//---------------------------------------------------------------------------------------------------------------
//
//  HAUD 2025.03.31
//
//  - EXAMPLE for top level procedures
//    - transport layer
//    - Collector layer
//    - process layer
//
//  - rewrite/change/discard as you require for your application
//
//  - this function block is NOT intended for direct use outside the scope of this example
//  - maybe the command mechanics are useful for your application
//
//---------------------------------------------------------------------------------------------------------------
FUNCTION_BLOCK fb_Application
VAR
  _eCheck                       : E_APP_CHECK;
  _eInit                        : E_PROGRESS;

  _Ctrl                         : REFERENCE TO ST_APP_CTRL;
  _State                        : REFERENCE TO ST_APP_STATE;

  _eResult                      : E_PROGRESS;

  _eCmd,
  _eCmdOld                      : E_INSTANCE_CMD;
  _eState                       : E_INSTANCE_STATE;

  // Transport Ctrl/State
  _XtsTransportCtrl             : REFERENCE TO ST_XTS_TRANSPORT_CTRL;
  _XtsTransportState            : REFERENCE TO ST_XTS_TRANSPORT_STATE;

  _InstanceCtrl                 : REFERENCE TO ARRAY[1..MAX_PROCESS] OF ST_INSTANCE_CTRL;
  _InstanceState                : REFERENCE TO ARRAY[1..MAX_PROCESS] OF ST_INSTANCE_STATE;
  
  _ItfProcessCollector          : REFERENCE TO ARRAY[1..MAX_PROCESS] OF I_ProcessCollector;

  _ItfProcessList               : REFERENCE TO ARRAY[1..MAX_PROCESS] OF I_Process_LinkedList;

  // timers for this example
  _tonProcess                   : ARRAY[1..MAX_PROCESS] OF Tc2_Standard.TON;
  _tProcess                     : ARRAY[1..MAX_PROCESS] OF TIME;


  _stMsg                        : ST_Message;
  _MessageLevel                 : E_MessageType;

  // ListData()
  _nLoadCaseOld,
  _nLoadCase                    : UINT := 0; // 0 = fully loaded, 2 = mod 5 missing 1, 1 = missing up to 11

  // Work()
  _bSingleOutput                : BOOL;
  _bWriteTimeVariant            : BOOL;
  _nTimeVariant                 : UINT;

  _sAppState                    : STRING;
END_VAR

IF NOT Check() THEN RETURN; END_IF
//-----------------------------------------------------------------------------
//-----------------------------------------------------------------------------
// set message device
//-----------------------------------------------------------------------------
_stMsg.eDevice                  := e_Device.Application;

_eCmd                           := _Ctrl.Cmd;
// check for command change
// get state for cmd
IF (_eCmd <> _eCmdOld)
THEN
  _eState                       := Cmd(_eCmd);
  _eCmdOld                      := _eCmd;
END_IF

CASE _eResult
OF
  E_PROGRESS.PROGRESS_INVALID:
    _State.AppState             := TO_UINT(_eResult);

  E_PROGRESS.PROGRESS_ERROR:
    _State.AppState             := _eState + E_PROGRESS.PROGRESS_ERROR;

  E_PROGRESS.PROGRESS_DONE:
    _State.AppState             := _eState + E_PROGRESS.PROGRESS_DONE;

    IF (_XtsTransportState.GroupInfo.GroupErrorStop) OR
       (_XtsTransportState.GroupInfo.GroupError)     OR
       NOT (_XtsTransportState.XpuInfo.AllPositionsValid)
    THEN
      _eResult                  := E_PROGRESS.PROGRESS_ERROR;
    END_IF
ELSE
  _State.AppState               := _eState + _eResult;

  CASE _eState
  OF
    E_INSTANCE_STATE.INIT:
      _eInit := _eResult        := Init(TRUE);

    E_INSTANCE_STATE.DISABLED:
      _eResult                  := Disable(TRUE);
  
    E_INSTANCE_STATE.ENABLED:
      IF NOT (_XtsTransportState.XpuState.DcLink) OR
         NOT (_XtsTransportState.XpuInfo.AllPositionsValid)
      THEN
        _eResult                := E_PROGRESS.PROGRESS_ERROR;
      ELSE
        _eResult                := Enable(TRUE);
      END_IF

    E_INSTANCE_STATE.WORKING:
      IF NOT (_XtsTransportState.XpuState.DcLink) OR
         NOT (_XtsTransportState.XpuInfo.AllPositionsValid)
      THEN
        _eResult                := E_PROGRESS.PROGRESS_ERROR;
      ELSE
        _eResult                := Work(TRUE);
      END_IF

    E_INSTANCE_STATE.PROCEEDING:
      IF NOT (_XtsTransportState.XpuState.DcLink) OR
         NOT (_XtsTransportState.XpuInfo.AllPositionsValid)
      THEN
        _eResult                := E_PROGRESS.PROGRESS_ERROR;
      ELSE
        _eResult                := Proceed(TRUE);
      END_IF

    E_INSTANCE_STATE.FINISH:
      IF NOT (_XtsTransportState.XpuState.DcLink) OR
         NOT (_XtsTransportState.XpuInfo.AllPositionsValid)
      THEN
        _eResult                := E_PROGRESS.PROGRESS_ERROR;
      ELSE
        _eResult                := Finish(TRUE);
      END_IF

    E_INSTANCE_STATE.CLEARED:
      _eResult                  := Clear(TRUE);


  ELSE
    _eResult                    := E_PROGRESS.PROGRESS_INVALID;
  END_CASE

END_CASE
_State.XtsTransportState        REF= _XtsTransportState;
_State.InstanceStates           REF= _InstanceState;


//IF _bWriteTimeVariant
//THEN
  _bWriteTimeVariant            := FALSE;

  CASE _nTimeVariant
  OF
    0:
      _tProcess[E_INSTANCE.INFEED]           := T#800MS;
      _tProcess[E_INSTANCE.OUTFEED_ROBOT_R1] := T#800MS;
      _tProcess[E_INSTANCE.OUTFEED_ROBOT_R2] := T#800MS;
    1:
      _tProcess[E_INSTANCE.INFEED]           := T#600MS;
      _tProcess[E_INSTANCE.OUTFEED_ROBOT_R1] := T#800MS;
      _tProcess[E_INSTANCE.OUTFEED_ROBOT_R2] := T#800MS;
    2:
      _tProcess[E_INSTANCE.INFEED]           := T#600MS;
      _tProcess[E_INSTANCE.OUTFEED_ROBOT_R1] := T#700MS;
      _tProcess[E_INSTANCE.OUTFEED_ROBOT_R2] := T#700MS;
    3:
      _tProcess[E_INSTANCE.INFEED]           := T#700MS;
      _tProcess[E_INSTANCE.OUTFEED_ROBOT_R1] := T#800MS;
      _tProcess[E_INSTANCE.OUTFEED_ROBOT_R2] := T#800MS;
    4:
      _tProcess[E_INSTANCE.INFEED]           := T#500MS;
      _tProcess[E_INSTANCE.OUTFEED_ROBOT_R1] := T#800MS;
      _tProcess[E_INSTANCE.OUTFEED_ROBOT_R2] := T#800MS;
    5:
      _tProcess[E_INSTANCE.INFEED]           := T#450MS;
      _tProcess[E_INSTANCE.OUTFEED_ROBOT_R1] := T#600MS;
      _tProcess[E_INSTANCE.OUTFEED_ROBOT_R2] := T#600MS;
  ELSE
      _tProcess[E_INSTANCE.INFEED]           := T#800MS;
      _tProcess[E_INSTANCE.OUTFEED_ROBOT_R1] := T#800MS;
      _tProcess[E_INSTANCE.OUTFEED_ROBOT_R2] := T#800MS;
  END_CASE
//END_IF

_sAppState := TO_STRING(_State.AppState);

METHOD Check : BOOL // call this method in the extending/inheriting class
VAR
  _nIdx       : E_INSTANCE;
END_VAR
//-----------------------------------------------------------------------------
//-----------------------------------------------------------------------------
// reference checks
//-----------------------------------------------------------------------------
IF NOT __ISVALIDREF(_Ctrl)
THEN
  _eCheck                   := E_APP_CHECK.INVALID_CTRL_POINTER;
  RETURN;
END_IF

IF NOT __ISVALIDREF(_State)
THEN
  _eCheck                   := E_APP_CHECK.INVALID_STATE_POINTER;
  RETURN;
END_IF

IF NOT __ISVALIDREF(_XtsTransportCtrl)
THEN
  _eCheck                   := E_APP_CHECK.INVALID_TRANSPORT_CTRL_POINTER;
  RETURN;
END_IF

IF NOT __ISVALIDREF(_XtsTransportState)
THEN
  _eCheck                   := E_APP_CHECK.INVALID_TRANSPORT_STATE_POINTER;
  RETURN;
END_IF

IF NOT __ISVALIDREF(_InstanceCtrl)
THEN
  _eCheck                   := E_APP_CHECK.INVALID_INSTANCE_CONTROL_REFERENCE;
  RETURN;
END_IF

IF NOT __ISVALIDREF(_InstanceState)
THEN
  _eCheck                   := E_APP_CHECK.INVALID_INSTANCE_STATE_REFERENCE;
  RETURN;
END_IF
IF NOT __ISVALIDREF(_ItfProcessCollector)
THEN
  _eCheck                   := E_APP_CHECK.INVALID_COLLECTOR_INTERFACE;
  RETURN;
END_IF
IF NOT __ISVALIDREF(_ItfProcessList)
THEN
  _eCheck                   := E_APP_CHECK.INVALID_PROCESS_LIST_INTERFACE;
  RETURN;
END_IF
//-----------------------------------------------------------------------------
//-----------------------------------------------------------------------------
// interface checks
//-----------------------------------------------------------------------------
FOR _nIdx := 1 TO MAX_PROCESS
DO
  IF NOT (_ItfProcessCollector[_nIdx] <> 0) 
  THEN
    _eCheck                 := E_APP_CHECK.INVALID_COLLECTOR_INTERFACE;
    RETURN;
  END_IF
  
  IF NOT (_ItfProcessCollector[_nIdx].ProcessId > 0)
  THEN
    _eCheck                 := E_APP_CHECK.INVALID_PROCESS_LIST_INTERFACE;
    RETURN;
  END_IF
END_FOR
//-----------------------------------------------------------------------------
//-----------------------------------------------------------------------------
_eCheck                     := E_APP_CHECK.CHECK_DONE;
Check                       := TRUE;
END_METHOD

METHOD Clear : E_PROGRESS
VAR_INPUT
  Execute     : BOOL;
END_VAR
VAR_INST
  _nErrorId   : UDINT;
  _eState     : E_PROGRESS;

  _eInstance  : E_INSTANCE;
END_VAR
//-----------------------------------------------------------------------------
IF NOT Execute 
THEN 
	_eState                                         := E_PROGRESS.PROGRESS_INIT; 
END_IF 
//-----------------------------------------------------------------------------
IF NOT Check() 
THEN 
	Clear                                            := E_PROGRESS.PROGRESS_ERROR; 
	RETURN; 
END_IF
//-----------------------------------------------------------------------------
//-----------------------------------------------------------------------------
CASE _eState
OF
  //---------------------------------------------------------------------------------------------------------------
  //---------------------------------------------------------------------------------------------------------------
  E_PROGRESS.PROGRESS_INIT:                   // startup procedure for your application
    IF Execute
    THEN
      ListData(FALSE, TRUE);
      _eState                                             := E_PROGRESS.PROGRESS_BUSY;
  
      FOR _eInstance := E_INSTANCE.BUFFER_INFEED TO E_INSTANCE.SENDER_BUFFER_INFEED
      DO
        _InstanceCtrl[_eInstance].Cmd                     := E_INSTANCE_CMD.NULL;
      END_FOR
  
      IF (_MessageLevel > E_MessageType.eMessageError)
      THEN
        _stMsg.eType                                      := E_MessageType.eMessageInfo;
        _stMsg.eSubdevice                                 := e_Subdevice.Application_Clear;
        _stMsg.iErrorNumber                               := 0;
        _stMsg.sText                                      := concat(TO_STRING(_eState), ': ');
        f_MessageSet(_stMsg);
      END_IF
    END_IF

  //---------------------------------------------------------------------------------------------------------------
  //---------------------------------------------------------------------------------------------------------------
  E_PROGRESS.PROGRESS_BUSY:
    ListData(FALSE, FALSE);
    _InstanceCtrl[E_INSTANCE.BUFFER_INFEED].Cmd           := E_INSTANCE_CMD.INIT;
    //-----------------------------------------------------------------------------------
    CASE _InstanceState[E_INSTANCE.BUFFER_INFEED].State
    OF
      E_INSTANCE_STATE.DISABLED:
        CASE _InstanceState[E_INSTANCE.BUFFER_INFEED].Progress
        OF
          E_PROGRESS.PROGRESS_BUSY:           // check for startup to be done
            _InstanceCtrl[E_INSTANCE.BUFFER_INFEED].Cmd   := E_INSTANCE_CMD.DISABLE;
            _eState                                       := E_PROGRESS.PROGRESS_PREPARE; // go check next insatnce

            IF (_MessageLevel > E_MessageType.eMessageError)
            THEN
              _stMsg.eType          := E_MessageType.eMessageInfo;
              _stMsg.eSubdevice     := e_Subdevice.Application_Clear;
              _stMsg.iErrorNumber   := 0;
              _stMsg.sText          := concat(TO_STRING(E_INSTANCE.BUFFER_INFEED), ': cleared');
              f_MessageSet(_stMsg);
            END_IF
        END_CASE
    END_CASE

  //---------------------------------------------------------------------------------------------------------------
  //---------------------------------------------------------------------------------------------------------------
  E_PROGRESS.PROGRESS_PREPARE:
    _InstanceCtrl[E_INSTANCE.INFEED].Cmd                  := E_INSTANCE_CMD.INIT;
    //-----------------------------------------------------------------------------------
    CASE _InstanceState[E_INSTANCE.INFEED].State
    OF
      E_INSTANCE_STATE.DISABLED:
        CASE _InstanceState[E_INSTANCE.INFEED].Progress
        OF
          E_PROGRESS.PROGRESS_BUSY:           // check for startup to be done
          _InstanceCtrl[E_INSTANCE.INFEED].Cmd            := E_INSTANCE_CMD.DISABLE;
          _eState                                         := E_PROGRESS.PROGRESS_STARTUP; // go check next insatnce

          IF (_MessageLevel > E_MessageType.eMessageError)
          THEN
            _stMsg.eType          := E_MessageType.eMessageInfo;
            _stMsg.eSubdevice     := e_Subdevice.Application_Clear;
            _stMsg.iErrorNumber   := 0;
            _stMsg.sText          := concat(TO_STRING(E_INSTANCE.INFEED), ': cleared');
            f_MessageSet(_stMsg);
          END_IF
        END_CASE
    END_CASE

  //---------------------------------------------------------------------------------------------------------------
  //---------------------------------------------------------------------------------------------------------------
  E_PROGRESS.PROGRESS_STARTUP:
    _InstanceCtrl[E_INSTANCE.BUFFER_OUTFEED].Cmd    := E_INSTANCE_CMD.INIT;
    //-----------------------------------------------------------------------------------
    CASE _InstanceState[E_INSTANCE.BUFFER_OUTFEED].State
    OF
      E_INSTANCE_STATE.DISABLED:
        CASE _InstanceState[E_INSTANCE.BUFFER_OUTFEED].Progress
        OF
          E_PROGRESS.PROGRESS_BUSY:           // check for startup to be done
          _InstanceCtrl[E_INSTANCE.BUFFER_OUTFEED].Cmd   := E_INSTANCE_CMD.DISABLE;
          _eState                                         := E_PROGRESS.PROGRESS_CHECK; // go check next insatnce

          IF (_MessageLevel > E_MessageType.eMessageError)
          THEN
            _stMsg.eType          := E_MessageType.eMessageInfo;
            _stMsg.eSubdevice     := e_Subdevice.Application_Clear;
            _stMsg.iErrorNumber   := 0;
            _stMsg.sText          := concat(TO_STRING(E_INSTANCE.BUFFER_OUTFEED), ': cleared');
            f_MessageSet(_stMsg);
          END_IF
        END_CASE
    END_CASE

  //---------------------------------------------------------------------------------------------------------------
  //---------------------------------------------------------------------------------------------------------------
  E_PROGRESS.PROGRESS_CHECK:
    _InstanceCtrl[E_INSTANCE.OUTFEED_ROBOT_R1].Cmd        := E_INSTANCE_CMD.INIT;
    //-----------------------------------------------------------------------------------
    CASE _InstanceState[E_INSTANCE.OUTFEED_ROBOT_R1].State
    OF
      E_INSTANCE_STATE.DISABLED:
        CASE _InstanceState[E_INSTANCE.OUTFEED_ROBOT_R1].Progress
        OF
          E_PROGRESS.PROGRESS_BUSY:           // check for startup to be done
          _InstanceCtrl[E_INSTANCE.OUTFEED_ROBOT_R1].Cmd  := E_INSTANCE_CMD.DISABLE;
          _eState                                         := E_PROGRESS.PROGRESS_OCCUPIED; // go check next insatnce

          IF (_MessageLevel > E_MessageType.eMessageError)
          THEN
            _stMsg.eType          := E_MessageType.eMessageInfo;
            _stMsg.eSubdevice     := e_Subdevice.Application_Clear;
            _stMsg.iErrorNumber   := 0;
            _stMsg.sText          := concat(TO_STRING(E_INSTANCE.OUTFEED_ROBOT_R1), ': cleared');
            f_MessageSet(_stMsg);
          END_IF
        END_CASE
    END_CASE

  //---------------------------------------------------------------------------------------------------------------
  //---------------------------------------------------------------------------------------------------------------
  E_PROGRESS.PROGRESS_OCCUPIED:
    _InstanceCtrl[E_INSTANCE.OUTFEED_ROBOT_R2].Cmd        := E_INSTANCE_CMD.INIT;
    //-----------------------------------------------------------------------------------
    CASE _InstanceState[E_INSTANCE.OUTFEED_ROBOT_R2].State
    OF
      E_INSTANCE_STATE.DISABLED:
        CASE _InstanceState[E_INSTANCE.OUTFEED_ROBOT_R2].Progress
        OF
          E_PROGRESS.PROGRESS_BUSY:           // check for startup to be done
          _InstanceCtrl[E_INSTANCE.OUTFEED_ROBOT_R2].Cmd  := E_INSTANCE_CMD.DISABLE;
          _eState                                         := E_PROGRESS.PROGRESS_WORKING; // go check next insatnce

          IF (_MessageLevel > E_MessageType.eMessageError)
          THEN
            _stMsg.eType          := E_MessageType.eMessageInfo;
            _stMsg.eSubdevice     := e_Subdevice.Application_Clear;
            _stMsg.iErrorNumber   := 0;
            _stMsg.sText          := concat(TO_STRING(E_INSTANCE.OUTFEED_ROBOT_R2), ': cleared');
            f_MessageSet(_stMsg);
          END_IF
        END_CASE
    END_CASE

  //---------------------------------------------------------------------------------------------------------------
  //---------------------------------------------------------------------------------------------------------------
  E_PROGRESS.PROGRESS_WORKING:
    _InstanceCtrl[E_INSTANCE.SENDER_FAST].Cmd             := E_INSTANCE_CMD.INIT;
    //-----------------------------------------------------------------------------------
    CASE _InstanceState[E_INSTANCE.SENDER_FAST].State
    OF
      E_INSTANCE_STATE.DISABLED:
        CASE _InstanceState[E_INSTANCE.SENDER_FAST].Progress
        OF
          E_PROGRESS.PROGRESS_BUSY:           // check for startup to be done
          _InstanceCtrl[E_INSTANCE.SENDER_FAST].Cmd       := E_INSTANCE_CMD.DISABLE;
          _eState                                         := E_PROGRESS.PROGRESS_STILL_WORKING; // go check next insatnce

          IF (_MessageLevel > E_MessageType.eMessageError)
          THEN
            _stMsg.eType          := E_MessageType.eMessageInfo;
            _stMsg.eSubdevice     := e_Subdevice.Application_Clear;
            _stMsg.iErrorNumber   := 0;
            _stMsg.sText          := concat(TO_STRING(E_INSTANCE.SENDER_FAST), ': cleared');
            f_MessageSet(_stMsg);
          END_IF
        END_CASE
    END_CASE

  //---------------------------------------------------------------------------------------------------------------
  //---------------------------------------------------------------------------------------------------------------
  E_PROGRESS.PROGRESS_STILL_WORKING:
    _InstanceCtrl[E_INSTANCE.SENDER_BUFFER_INFEED].Cmd    := E_INSTANCE_CMD.INIT;
    //-----------------------------------------------------------------------------------
    CASE _InstanceState[E_INSTANCE.SENDER_BUFFER_INFEED].State
    OF
      E_INSTANCE_STATE.DISABLED:
        CASE _InstanceState[E_INSTANCE.SENDER_BUFFER_INFEED].Progress
        OF
          E_PROGRESS.PROGRESS_BUSY:           // check for startup to be done
          _InstanceCtrl[E_INSTANCE.SENDER_BUFFER_INFEED].Cmd    := E_INSTANCE_CMD.DISABLE;
          _eState                                         := E_PROGRESS.PROGRESS_DONE;

          IF (_MessageLevel > E_MessageType.eMessageError)
          THEN
            _stMsg.eType          := E_MessageType.eMessageInfo;
            _stMsg.eSubdevice     := e_Subdevice.Application_Clear;
            _stMsg.iErrorNumber   := 0;
            _stMsg.sText          := concat(TO_STRING(E_INSTANCE.SENDER_BUFFER_INFEED), ': cleared');
            f_MessageSet(_stMsg);
          END_IF

          IF (_MessageLevel > E_MessageType.eMessageError)
          THEN
            _stMsg.eType          := E_MessageType.eMessageInfo;
            _stMsg.eSubdevice     := e_Subdevice.Application_Clear;
            _stMsg.iErrorNumber   := 0;
            _stMsg.sText          := concat(TO_STRING(_eState), ': ');
            f_MessageSet(_stMsg);
          END_IF
        END_CASE
    END_CASE
END_CASE
//-----------------------------------------------------------------------------
//-----------------------------------------------------------------------------

Clear                                              := _eState;
END_METHOD

METHOD PRIVATE Cmd : E_INSTANCE_STATE
VAR_INPUT
  Command   : E_INSTANCE_CMD;
END_VAR
VAR_INST
  _eRslt    : E_PROGRESS;
  _eState   : E_INSTANCE_STATE;
END_VAR
IF NOT Check() THEN RETURN; END_IF


CASE Command
OF
  E_INSTANCE_CMD.NULL:  // clear all method calls
    _eState               := E_INSTANCE_STATE.NULL;
    _eRslt                := Init    (FALSE);
    _eRslt                := Disable (FALSE);
    _eRslt                := Enable  (FALSE);
    _eRslt                := Work    (FALSE);
    _eRslt                := Proceed (FALSE);
    _eRslt                := Finish  (FALSE);
    _eRslt                := Clear   (FALSE);

  E_INSTANCE_CMD.INIT:  // clear methods for initialization
    _eState               := E_INSTANCE_STATE.INIT;
    _eResult              := Init(FALSE);

ELSE
  IF NOT (_eInit = E_PROGRESS.PROGRESS_DONE)
  THEN
    // no init, no further commands possible
    _eState               := E_INSTANCE_STATE.INVALID;
  ELSE
    CASE Command
    OF
      E_INSTANCE_CMD.DISABLE:
        _eState           := E_INSTANCE_STATE.DISABLED;
        _eResult          := Disable (FALSE);

      E_INSTANCE_CMD.ENABLE:
        _eState           := E_INSTANCE_STATE.ENABLED;
        _eResult          := Enable  (FALSE);

      E_INSTANCE_CMD.WORK:
        _eState           := E_INSTANCE_STATE.WORKING;
        _eResult          := Work    (FALSE);

      E_INSTANCE_CMD.PROCEED:
        _eState           := E_INSTANCE_STATE.PROCEEDING;
        _eResult          := Proceed (FALSE);

      E_INSTANCE_CMD.FINISH:
        _eState           := E_INSTANCE_STATE.FINISH;
        _eResult          := Finish  (FALSE);

      E_INSTANCE_CMD.CLEAR:
        _eState           := E_INSTANCE_STATE.CLEARED;
        _eResult          := Clear   (FALSE);

    ELSE
        _eState           := E_INSTANCE_STATE.INVALID;
    END_CASE
  END_IF
END_CASE

Cmd                       := _eState;
END_METHOD

PROPERTY CollectorInterface : REFERENCE TO ARRAY[1..MAX_PROCESS] OF I_ProcessCollector
SET
_ItfProcessCollector REF= CollectorInterface;
END_SET
END_PROPERTY

PROPERTY Ctrl : REFERENCE TO ST_APP_CTRL
SET
_Ctrl REF= Ctrl;
END_SET
END_PROPERTY

METHOD Disable : E_PROGRESS // RemoveAllAxis from CA Group, disable CA Group, disable all movers
VAR_INPUT
  Execute     : BOOL;
END_VAR
VAR_INST
  _nErrorId   : UDINT;
  _eState     : E_PROGRESS;
END_VAR
//-----------------------------------------------------------------------------
IF NOT Execute 
THEN 
	_eState                       := E_PROGRESS.PROGRESS_INIT; 
END_IF 
//-----------------------------------------------------------------------------
IF NOT Check() 
THEN 
	Disable                       := E_PROGRESS.PROGRESS_ERROR; 
	RETURN; 
END_IF
//-----------------------------------------------------------------------------
//-----------------------------------------------------------------------------
CASE _eState
OF
  E_PROGRESS.PROGRESS_INIT:
    IF Execute
    THEN
      _nErrorId                 := 0;

      _XtsTransportCtrl.Cmd     := E_XTS_TRANSPORT_CTRL.CMD_NULL;
      _eState                   := E_PROGRESS.PROGRESS_BUSY;

      IF (_MessageLevel > E_MessageType.eMessageError)
      THEN
        _stMsg.eType            := E_MessageType.eMessageInfo;
        _stMsg.eSubdevice       := e_Subdevice.Application_Disable;
        _stMsg.iErrorNumber     := 0;
        _stMsg.sText            := concat(TO_STRING(_eState), ': ');
        f_MessageSet(_stMsg);
      END_IF
    END_IF

  E_PROGRESS.PROGRESS_BUSY:
    _XtsTransportCtrl.Cmd       := E_XTS_TRANSPORT_CTRL.CMD_GROUP_CLEAR; 
    _eState                     := E_PROGRESS.PROGRESS_PREPARE;
END_CASE
//-----------------------------------------------------------------------------
//-----------------------------------------------------------------------------
CASE _eState
OF
  E_PROGRESS.PROGRESS_PREPARE:
    IF (_XtsTransportState.State = E_XTS_TRANSPORT_STATE.TRANSPORT_GROUP_CLEAR + E_PROGRESS.PROGRESS_ERROR)
    THEN
      _eState                   := E_PROGRESS.PROGRESS_BUSY;
      _XtsTransportCtrl.Cmd     := E_XTS_TRANSPORT_CTRL.CMD_NULL;

      _nErrorId                 := _XtsTransportState.GroupInfo.GroupErrorId; 

    ELSIF (_XtsTransportState.State = E_XTS_TRANSPORT_STATE.TRANSPORT_GROUP_CLEAR + E_PROGRESS.PROGRESS_DONE)
    THEN
      _eState                   := E_PROGRESS.PROGRESS_STARTUP;

    END_IF
END_CASE
//-----------------------------------------------------------------------------
//-----------------------------------------------------------------------------
CASE _eState
OF
  E_PROGRESS.PROGRESS_STARTUP:
    _XtsTransportCtrl.Cmd       := E_XTS_TRANSPORT_CTRL.CMD_MOVER_DISABLE; 
    _eState                     := E_PROGRESS.PROGRESS_CHECK;
END_CASE
//-----------------------------------------------------------------------------
//-----------------------------------------------------------------------------
CASE _eState
OF
  E_PROGRESS.PROGRESS_CHECK:
    IF (_XtsTransportState.State = E_XTS_TRANSPORT_STATE.TRANSPORT_MOVER_DISABLE + E_PROGRESS.PROGRESS_ERROR)
    THEN
      _eState                   := E_PROGRESS.PROGRESS_ERROR;

    ELSIF (_XtsTransportState.State = E_XTS_TRANSPORT_STATE.TRANSPORT_MOVER_DISABLE + E_PROGRESS.PROGRESS_DONE)
    THEN
      _eState                   := E_PROGRESS.PROGRESS_DONE;

      IF (_MessageLevel > E_MessageType.eMessageError)
      THEN
        _stMsg.eType            := E_MessageType.eMessageInfo;
        _stMsg.eSubdevice       := e_Subdevice.Application_Disable;
        _stMsg.iErrorNumber     := 0;
        _stMsg.sText            := concat(TO_STRING(_eState), ': ');
        f_MessageSet(_stMsg);
      END_IF
    END_IF
END_CASE
//-----------------------------------------------------------------------------
//-----------------------------------------------------------------------------

Disable                         := _eState;
END_METHOD

METHOD Enable : E_PROGRESS // AddAllAxis to CA Group, Enable CA Group, Enable all movers
VAR_INPUT
  Execute     : BOOL;
END_VAR
VAR_INST
  _nErrorId   : UDINT;
  _eState     : E_PROGRESS;
END_VAR
//-----------------------------------------------------------------------------
IF NOT Execute 
THEN 
	_eState                       := E_PROGRESS.PROGRESS_INIT; 
END_IF 
//-----------------------------------------------------------------------------
IF NOT Check() 
THEN 
	Enable                        := E_PROGRESS.PROGRESS_ERROR; 
	RETURN; 
END_IF
//-----------------------------------------------------------------------------
//-----------------------------------------------------------------------------
CASE _eState
OF
  E_PROGRESS.PROGRESS_INIT:
    IF Execute
    THEN

      IF (GVL_APPLICATION.bOutput_R1R2)
      THEN
        MAIN_APP.ProcessInit_R1R2();
      ELSE
        MAIN_APP.ProcessInit_CLAMP();
      END_IF

      _nErrorId                 := 0;

      _XtsTransportCtrl.Cmd     := E_XTS_TRANSPORT_CTRL.CMD_NULL;
      _eState                   := E_PROGRESS.PROGRESS_BUSY;

      IF (_MessageLevel > E_MessageType.eMessageError)
      THEN
        _stMsg.eType            := E_MessageType.eMessageInfo;
        _stMsg.eSubdevice       := e_Subdevice.Application_Enable;
        _stMsg.iErrorNumber     := 0;
        _stMsg.sText            := concat(TO_STRING(_eState), ': ');
        f_MessageSet(_stMsg);
      END_IF
    END_IF

  E_PROGRESS.PROGRESS_BUSY:
    _XtsTransportCtrl.Cmd       := E_XTS_TRANSPORT_CTRL.CMD_GROUP_BUILD; 
    _eState                     := E_PROGRESS.PROGRESS_PREPARE;
END_CASE
//-----------------------------------------------------------------------------
//-----------------------------------------------------------------------------
CASE _eState
OF
  E_PROGRESS.PROGRESS_PREPARE:
    IF (_XtsTransportState.State = E_XTS_TRANSPORT_STATE.TRANSPORT_GROUP_BUILD + E_PROGRESS.PROGRESS_ERROR)
    THEN
      _eState                   := E_PROGRESS.PROGRESS_ERROR;
      _nErrorId                 := _XtsTransportState.GroupInfo.GroupErrorId; 

    ELSIF (_XtsTransportState.State = E_XTS_TRANSPORT_STATE.TRANSPORT_GROUP_BUILD + E_PROGRESS.PROGRESS_DONE)
    THEN
      _eState                   := E_PROGRESS.PROGRESS_STARTUP;
    END_IF
END_CASE
//-----------------------------------------------------------------------------
//-----------------------------------------------------------------------------
CASE _eState
OF
  E_PROGRESS.PROGRESS_STARTUP:
    _XtsTransportCtrl.Cmd       := E_XTS_TRANSPORT_CTRL.CMD_MOVER_ENABLE; 
    _eState                     := E_PROGRESS.PROGRESS_CHECK;
END_CASE
//-----------------------------------------------------------------------------
//-----------------------------------------------------------------------------
CASE _eState
OF
  E_PROGRESS.PROGRESS_CHECK:
    IF (_XtsTransportState.State = E_XTS_TRANSPORT_STATE.TRANSPORT_MOVER_ENABLE + E_PROGRESS.PROGRESS_ERROR)
    THEN
      _eState                   := E_PROGRESS.PROGRESS_ERROR;

    ELSIF (_XtsTransportState.State = E_XTS_TRANSPORT_STATE.TRANSPORT_MOVER_ENABLE + E_PROGRESS.PROGRESS_DONE)
    THEN
      _eState                   := E_PROGRESS.PROGRESS_OCCUPIED;
    END_IF
END_CASE
//-----------------------------------------------------------------------------
//-----------------------------------------------------------------------------
CASE _eState
OF
  E_PROGRESS.PROGRESS_OCCUPIED:
    _XtsTransportCtrl.Cmd       := E_XTS_TRANSPORT_CTRL.CMD_GROUP_ENABLE; 
    _eState                     := E_PROGRESS.PROGRESS_WORKING;
END_CASE
//-----------------------------------------------------------------------------
//-----------------------------------------------------------------------------
CASE _eState
OF
  E_PROGRESS.PROGRESS_WORKING:
    IF (_XtsTransportState.State = E_XTS_TRANSPORT_STATE.TRANSPORT_GROUP_ENABLE + E_PROGRESS.PROGRESS_ERROR)
    THEN
      _eState                   := E_PROGRESS.PROGRESS_ERROR;

    ELSIF (_XtsTransportState.State = E_XTS_TRANSPORT_STATE.TRANSPORT_GROUP_ENABLE + E_PROGRESS.PROGRESS_DONE)
    THEN
      _eState                   := E_PROGRESS.PROGRESS_DONE;

      IF (_MessageLevel > E_MessageType.eMessageError)
      THEN
        _stMsg.eType            := E_MessageType.eMessageInfo;
        _stMsg.eSubdevice       := e_Subdevice.Application_Enable;
        _stMsg.iErrorNumber     := 0;
        _stMsg.sText            := concat(TO_STRING(_eState), ': ');
        f_MessageSet(_stMsg);
      END_IF
    END_IF
END_CASE
//-----------------------------------------------------------------------------
//-----------------------------------------------------------------------------

Enable                          := _eState;
END_METHOD

METHOD Finish : E_PROGRESS
VAR_INPUT
  Execute     : BOOL;
END_VAR
VAR_INST
  _nErrorId               : UDINT;
  _eState                 : E_PROGRESS;

  _nExp                   : BYTE;
  _WriteData              : ST_PROCESS_DATA;
  _ListResult             : ST_PROCESS_LIST_RESULT;

  _eInst                  : E_INSTANCE;
  _bDbg : BOOL;
  {attribute 'displaymode':='bin'}
  _wDisable               : T_PROCESS;

  _nSwitch                : UINT;
  _TransportState         : E_XTS_TRANSPORT_STATE;
  _JobResult              : E_PROGRESS;
END_VAR
//-----------------------------------------------------------------------------
IF NOT Execute 
THEN 
	_eState                       := E_PROGRESS.PROGRESS_INIT; 
END_IF 
//-----------------------------------------------------------------------------
IF NOT Check() 
THEN 
	Finish                        := E_PROGRESS.PROGRESS_ERROR; 
	RETURN; 
END_IF
//-----------------------------------------------------------------------------
//-----------------------------------------------------------------------------
CASE _eState
OF
  E_PROGRESS.PROGRESS_INIT:
    IF Execute
    THEN
      _nErrorId                 := 0;
      _JobResult                := ListData(TRUE, FALSE);     // reset simulated transfersystem

      IF NOT (_XtsTransportState.GroupInfo.GroupErrorStop)
      THEN
        _eState                 := E_PROGRESS.PROGRESS_BUSY;

        IF (_MessageLevel > E_MessageType.eMessageError)
        THEN
          _stMsg.eType          := E_MessageType.eMessageInfo;
          _stMsg.eSubdevice     := e_Subdevice.Application_Finish;
          _stMsg.iErrorNumber   := 0;
          _stMsg.sText          := concat(TO_STRING(_eState), ': ');
          f_MessageSet(_stMsg);
        END_IF
      ELSE
        _nErrorId               := _XtsTransportState.GroupInfo.GroupErrorId;
        _eState                 := E_PROGRESS.PROGRESS_ERROR;

        _stMsg.eType            := E_MessageType.eMessageError;
        _stMsg.eSubdevice       := e_Subdevice.Application_Finish;
        _stMsg.iErrorNumber     := _nErrorId;
        _stMsg.sText            := concat(TO_STRING(_eState), ': ');
        _stMsg.sText            := concat(_stMsg.sText, ' CaGroup ErrorStop');
        f_MessageSet(_stMsg);
      END_IF
    END_IF


  E_PROGRESS.PROGRESS_BUSY:
    IF (_XtsTransportState.State = E_XTS_TRANSPORT_STATE.TRANSPORT_START   + E_PROGRESS.PROGRESS_ERROR) OR
       (_XtsTransportState.State = E_XTS_TRANSPORT_STATE.TRANSPORT_RESTART + E_PROGRESS.PROGRESS_ERROR)
    THEN
      _eState                   := E_PROGRESS.PROGRESS_ERROR;

      _stMsg.eType              := E_MessageType.eMessageError;
      _stMsg.eSubdevice         := e_Subdevice.Application_Finish;
      _stMsg.iErrorNumber       := 0;
      _stMsg.sText              := concat(TO_STRING(_eState), ': ');
      _stMsg.sText              := concat(_stMsg.sText, TO_STRING(_XtsTransportState.State MOD E_PROGRESS.PROGRESS_ERROR));
      f_MessageSet(_stMsg);

    ELSIF (_XtsTransportState.State = E_XTS_TRANSPORT_STATE.TRANSPORT_START   + E_PROGRESS.PROGRESS_DONE) OR
          (_XtsTransportState.State = E_XTS_TRANSPORT_STATE.TRANSPORT_RESTART + E_PROGRESS.PROGRESS_DONE)
    THEN
      _JobResult                := ListData(FALSE, FALSE);     // stop simulated transfersystem
      _wDisable                 := 0;
      _eState                   := E_PROGRESS.PROGRESS_PREPARE;

      IF (_MessageLevel > E_MessageType.eMessageError)
      THEN
        _stMsg.eType            := E_MessageType.eMessageInfo;
        _stMsg.eSubdevice       := e_Subdevice.Application_Finish;
        _stMsg.iErrorNumber     := 0;
        _stMsg.sText            := concat(TO_STRING(_eState), ': ');
        _stMsg.sText            := concat(_stMsg.sText, TO_STRING(_XtsTransportState.State MOD E_PROGRESS.PROGRESS_DONE));
        f_MessageSet(_stMsg);
      END_IF
    END_IF
END_CASE
//-----------------------------------------------------------------------------
//-----------------------------------------------------------------------------
CASE _eState
OF
  E_PROGRESS.PROGRESS_PREPARE:  // SENDER_BUFFER_INFEED sends movers to BUFFER_INFEED
                                //  - this instance has to stop first
    CASE _InstanceState[E_INSTANCE.SENDER_BUFFER_INFEED].State
    OF
    E_INSTANCE_STATE.DISABLED:

      CASE _InstanceState[E_INSTANCE.SENDER_BUFFER_INFEED].Progress
      OF
      E_PROGRESS.PROGRESS_BUSY,
      E_PROGRESS.PROGRESS_PREPARE:
        _eState                                               := E_PROGRESS.PROGRESS_STARTUP;
        _InstanceCtrl[E_INSTANCE.SENDER_BUFFER_INFEED].Cmd    := E_INSTANCE_CMD.DISABLE;
  
        _wDisable                                             := _ItfProcessCollector[E_INSTANCE.SENDER_BUFFER_INFEED].
                                                                 SetBit(_wDisable, TO_BYTE(E_INSTANCE.SENDER_BUFFER_INFEED-1));
        IF (_MessageLevel > E_MessageType.eMessageError)
        THEN
          _stMsg.eType                                        := E_MessageType.eMessageInfo;
          _stMsg.eSubdevice                                   := e_Subdevice.Application_Finish;
          _stMsg.iErrorNumber                                 := 0;
          _stMsg.sText                                        := concat(TO_STRING(E_INSTANCE.SENDER_BUFFER_INFEED), ': _wDisable  ');
          _stMsg.sText                                        := concat(_stMsg.sText, _ItfProcessCollector[E_INSTANCE.SENDER_BUFFER_INFEED].BitsToString(_wDisable));
          f_MessageSet(_stMsg);
        END_IF
      END_CASE
    END_CASE
END_CASE
//-----------------------------------------------------------------------------
//-----------------------------------------------------------------------------
CASE _eState
OF
  E_PROGRESS.PROGRESS_STARTUP:
    _JobResult                                                := ListData(FALSE, FALSE);     // stop simulated transfersystem

    CASE _InstanceState[E_INSTANCE.BUFFER_INFEED].State
    OF
    E_INSTANCE_STATE.DISABLED,
    E_INSTANCE_STATE.DETECTION:

      _eState                                                 := E_PROGRESS.PROGRESS_CHECK;
      _InstanceCtrl[E_INSTANCE.BUFFER_INFEED].Cmd             := E_INSTANCE_CMD.DISABLE;
  
      IF NOT (_ItfProcessCollector[E_INSTANCE.BUFFER_INFEED].GetBit(_wDisable, TO_BYTE(E_INSTANCE.BUFFER_INFEED-1)))
      THEN
        _wDisable                                             := _ItfProcessCollector[E_INSTANCE.BUFFER_INFEED].
                                                                 SetBit(_wDisable, TO_BYTE(E_INSTANCE.BUFFER_INFEED-1));
  
        IF (_MessageLevel > E_MessageType.eMessageError)
        THEN
          _stMsg.eType                                        := E_MessageType.eMessageInfo;
          _stMsg.eSubdevice                                   := e_Subdevice.Application_Finish;
          _stMsg.iErrorNumber                                 := 0;
          _stMsg.sText                                        := concat(TO_STRING(E_INSTANCE.BUFFER_INFEED), ': _wDisable  ');
          _stMsg.sText                                        := concat(_stMsg.sText, _ItfProcessCollector[E_INSTANCE.BUFFER_INFEED].BitsToString(_wDisable));
          f_MessageSet(_stMsg);
        END_IF
      END_IF

    E_INSTANCE_STATE.ENABLED:
      _InstanceCtrl[E_INSTANCE.BUFFER_INFEED].Cmd             := E_INSTANCE_CMD.DISABLE;


    E_INSTANCE_STATE.FINISH:
      CASE _InstanceState[E_INSTANCE.BUFFER_INFEED].Progress
      OF
        E_PROGRESS.PROGRESS_BUSY:
          _InstanceCtrl[E_INSTANCE.BUFFER_INFEED].Cmd         := E_INSTANCE_CMD.FINISH;

        E_PROGRESS.PROGRESS_OCCUPIED:
          _InstanceCtrl[E_INSTANCE.BUFFER_INFEED].Cmd         := E_INSTANCE_CMD.PROCEED;
      END_CASE
    END_CASE
END_CASE
//-----------------------------------------------------------------------------
//-----------------------------------------------------------------------------
CASE _eState
OF
  E_PROGRESS.PROGRESS_CHECK:
    CASE _InstanceState[E_INSTANCE.INFEED].State
    OF
    E_INSTANCE_STATE.DISABLED,
    E_INSTANCE_STATE.DETECTION:

      CASE _InstanceState[E_INSTANCE.INFEED].Progress
      OF
      E_PROGRESS.PROGRESS_BUSY:
          IF (_ItfProcessCollector[E_INSTANCE.BUFFER_INFEED].QueueProcessCount > 0)
          THEN
            _eState                                           := E_PROGRESS.PROGRESS_STARTUP;
            _InstanceCtrl[E_INSTANCE.INFEED].Cmd              := E_INSTANCE_CMD.ENABLE;

          ELSIF (_ItfProcessList[E_INSTANCE.INFEED].Count > 0)
          THEN
            _InstanceCtrl[E_INSTANCE.INFEED].Cmd              := E_INSTANCE_CMD.ENABLE;
          ELSE
            _eState                                           := E_PROGRESS.PROGRESS_OCCUPIED;
            _InstanceCtrl[E_INSTANCE.INFEED].Cmd              := E_INSTANCE_CMD.DISABLE;

            IF NOT (_ItfProcessCollector[E_INSTANCE.INFEED].GetBit(_wDisable, TO_BYTE(E_INSTANCE.INFEED-1)))
            THEN
              _wDisable                                       := _ItfProcessCollector[E_INSTANCE.INFEED].
                                                                   SetBit(_wDisable, TO_BYTE(E_INSTANCE.INFEED-1));

              IF (_MessageLevel > E_MessageType.eMessageError)
              THEN
                _stMsg.eType                                  := E_MessageType.eMessageInfo;
                _stMsg.eSubdevice                             := e_Subdevice.Application_Finish;
                _stMsg.iErrorNumber                           := 0;
                _stMsg.sText                                  := concat(TO_STRING(E_INSTANCE.INFEED), ': _wDisable ');
                _stMsg.sText                                  := concat(_stMsg.sText, _ItfProcessCollector[E_INSTANCE.INFEED].BitsToString(_wDisable));
                f_MessageSet(_stMsg);
              END_IF
            END_IF
          END_IF
      END_CASE

    E_INSTANCE_STATE.ENABLED:
      CASE _InstanceState[E_INSTANCE.INFEED].Progress
      OF
        E_PROGRESS.PROGRESS_OCCUPIED:
          _InstanceCtrl[E_INSTANCE.INFEED].Cmd                := E_INSTANCE_CMD.PROCEED;
      END_CASE


    E_INSTANCE_STATE.WORKING:
      CASE _InstanceState[E_INSTANCE.INFEED].Progress
      OF
        E_PROGRESS.PROGRESS_BUSY:
          _InstanceCtrl[E_INSTANCE.INFEED].Cmd                := E_INSTANCE_CMD.WORK;
          _tonProcess [E_INSTANCE.INFEED]
                                          (IN                 := FALSE, 
                                           PT                 := _tProcess[E_INSTANCE.INFEED]);
  
        E_PROGRESS.PROGRESS_CHECK:
          _tonProcess [E_INSTANCE.INFEED]
                                          (IN                 := TRUE, 
                                           PT                 := _tProcess[E_INSTANCE.INFEED]);
  
          IF _tonProcess [E_INSTANCE.INFEED].Q
          THEN
            _InstanceCtrl[E_INSTANCE.INFEED].Cmd              := E_INSTANCE_CMD.FINISH;
          END_IF
      END_CASE

    E_INSTANCE_STATE.FINISH:
      CASE _InstanceState[E_INSTANCE.INFEED].Progress
      OF
        E_PROGRESS.PROGRESS_BUSY:
          _InstanceCtrl[E_INSTANCE.INFEED].Cmd                := E_INSTANCE_CMD.FINISH;

        E_PROGRESS.PROGRESS_OCCUPIED:
          _InstanceCtrl[E_INSTANCE.INFEED].Cmd                := E_INSTANCE_CMD.PROCEED;
      END_CASE
    END_CASE

    CASE _InstanceState[E_INSTANCE.BUFFER_OUTFEED].State
    OF
    E_INSTANCE_STATE.DISABLED:

      CASE _InstanceState[E_INSTANCE.BUFFER_OUTFEED].Progress
      OF
      E_PROGRESS.PROGRESS_BUSY:
        _InstanceCtrl[E_INSTANCE.BUFFER_OUTFEED].Cmd    := E_INSTANCE_CMD.ENABLE;
      END_CASE

    E_INSTANCE_STATE.FINISH:
      CASE _InstanceState[E_INSTANCE.BUFFER_OUTFEED].Progress
      OF
        E_PROGRESS.PROGRESS_BUSY:
          _InstanceCtrl[E_INSTANCE.BUFFER_OUTFEED].Cmd  := E_INSTANCE_CMD.FINISH;

        E_PROGRESS.PROGRESS_OCCUPIED:
          _InstanceCtrl[E_INSTANCE.BUFFER_OUTFEED].Cmd  := E_INSTANCE_CMD.PROCEED;

        E_PROGRESS.PROGRESS_DONE:
          _InstanceCtrl[E_INSTANCE.BUFFER_OUTFEED].Cmd  := E_INSTANCE_CMD.DISABLE;
      END_CASE
    END_CASE

    CASE _InstanceState[E_INSTANCE.SENDER_FAST].State
    OF
      E_INSTANCE_STATE.DISABLED:
        CASE _InstanceState[E_INSTANCE.SENDER_FAST].Progress
        OF
          E_PROGRESS.PROGRESS_BUSY:
            IF NOT (_ItfProcessCollector[E_INSTANCE.OUTFEED_ROBOT_R1].QueueProcessCount < 12) OR 
               NOT (_ItfProcessCollector[E_INSTANCE.OUTFEED_ROBOT_R2].QueueProcessCount < 12)
            THEN
              _InstanceCtrl[E_INSTANCE.SENDER_FAST].Cmd       := E_INSTANCE_CMD.ENABLE;

            ELSIF (_ItfProcessCollector[E_INSTANCE.SENDER_FAST].QueueProcessCount > 0)
            THEN
              _InstanceCtrl[E_INSTANCE.SENDER_FAST].Cmd       := E_INSTANCE_CMD.ENABLE;
            ELSE
              _InstanceCtrl[E_INSTANCE.SENDER_FAST].Cmd       := E_INSTANCE_CMD.DISABLE;

              IF NOT (_ItfProcessCollector[E_INSTANCE.SENDER_FAST].GetBit(_wDisable, TO_BYTE(E_INSTANCE.SENDER_FAST-1)))
              THEN
                _wDisable                                     := _ItfProcessCollector[E_INSTANCE.SENDER_FAST].
                                                                 SetBit(_wDisable, TO_BYTE(E_INSTANCE.SENDER_FAST-1));
    
                IF (_MessageLevel > E_MessageType.eMessageError)
                THEN
                  _stMsg.eType                                := E_MessageType.eMessageInfo;
                  _stMsg.eSubdevice                           := e_Subdevice.Application_Finish;
                  _stMsg.iErrorNumber                         := 0;
                  _stMsg.sText                                := concat(TO_STRING(E_INSTANCE.SENDER_FAST), ': _wDisable ');
                  _stMsg.sText                                := concat(_stMsg.sText, _ItfProcessCollector[E_INSTANCE.SENDER_FAST].BitsToString(_wDisable));
                  f_MessageSet(_stMsg);
                END_IF
              END_IF
            END_IF
        END_CASE

      E_INSTANCE_STATE.FINISH:
        CASE _InstanceState[E_INSTANCE.SENDER_FAST].Progress
        OF
          E_PROGRESS.PROGRESS_BUSY:
            _InstanceCtrl[E_INSTANCE.SENDER_FAST].Cmd         := E_INSTANCE_CMD.FINISH;
        END_CASE
      END_CASE
END_CASE
//-----------------------------------------------------------------------------
//-----------------------------------------------------------------------------
CASE _eState
OF
  E_PROGRESS.PROGRESS_OCCUPIED:
    CASE _InstanceState[E_INSTANCE.BUFFER_OUTFEED].State
    OF
    E_INSTANCE_STATE.DISABLED:

      CASE _InstanceState[E_INSTANCE.BUFFER_OUTFEED].Progress
      OF
      E_PROGRESS.PROGRESS_BUSY:
        IF (_ItfProcessCollector[E_INSTANCE.INFEED].QueueProcessCount > 11)
        THEN
          _eState                                             := E_PROGRESS.PROGRESS_CHECK;
          _InstanceCtrl[E_INSTANCE.BUFFER_OUTFEED].Cmd  := E_INSTANCE_CMD.ENABLE;

        ELSIF (_ItfProcessCollector[E_INSTANCE.BUFFER_OUTFEED].QueueProcessCount > 0)
        THEN
          _InstanceCtrl[E_INSTANCE.BUFFER_OUTFEED].Cmd  := E_INSTANCE_CMD.ENABLE;
        ELSE
          _eState                                             := E_PROGRESS.PROGRESS_WORKING;
          _InstanceCtrl[E_INSTANCE.BUFFER_OUTFEED].Cmd  := E_INSTANCE_CMD.DISABLE;

            IF NOT (_ItfProcessCollector[E_INSTANCE.BUFFER_OUTFEED].GetBit(_wDisable, TO_BYTE(E_INSTANCE.BUFFER_OUTFEED-1)))
            THEN
              _wDisable                                       := _ItfProcessCollector[E_INSTANCE.BUFFER_OUTFEED].
                                                                   SetBit(_wDisable, TO_BYTE(E_INSTANCE.BUFFER_OUTFEED-1));

              IF (_MessageLevel > E_MessageType.eMessageError)
              THEN
                _stMsg.eType                                  := E_MessageType.eMessageInfo;
                _stMsg.eSubdevice                             := e_Subdevice.Application_Finish;
                _stMsg.iErrorNumber                           := 0;
                _stMsg.sText                                  := concat(TO_STRING(E_INSTANCE.BUFFER_OUTFEED), ': _wDisable ');
                _stMsg.sText                                  := concat(_stMsg.sText, _ItfProcessCollector[E_INSTANCE.BUFFER_OUTFEED].BitsToString(_wDisable));
                f_MessageSet(_stMsg);
              END_IF
            END_IF
        END_IF
      END_CASE

    E_INSTANCE_STATE.ENABLED:
      _InstanceCtrl[E_INSTANCE.BUFFER_OUTFEED].Cmd      := E_INSTANCE_CMD.DISABLE;


    E_INSTANCE_STATE.FINISH:
      CASE _InstanceState[E_INSTANCE.BUFFER_OUTFEED].Progress
      OF
        E_PROGRESS.PROGRESS_BUSY:
          _InstanceCtrl[E_INSTANCE.BUFFER_OUTFEED].Cmd  := E_INSTANCE_CMD.FINISH;

        E_PROGRESS.PROGRESS_OCCUPIED:
          _InstanceCtrl[E_INSTANCE.BUFFER_OUTFEED].Cmd  := E_INSTANCE_CMD.PROCEED;

        E_PROGRESS.PROGRESS_DONE:
          _InstanceCtrl[E_INSTANCE.BUFFER_OUTFEED].Cmd  := E_INSTANCE_CMD.DISABLE;
      END_CASE
    END_CASE
END_CASE
//-----------------------------------------------------------------------------
//-----------------------------------------------------------------------------
CASE _eState
OF
  E_PROGRESS.PROGRESS_WORKING:
    IF (_wDisable = EXPT(2, E_INSTANCE.SENDER_BUFFER_INFEED)-1)
    THEN
      _eState                                                 := E_PROGRESS.PROGRESS_STILL_WORKING;
    END_IF

    //-------------------------------------------------------------------------
    // E_INSTANCE.OUTFEED_ROBOT_R1
    //-------------------------------------------------------------------------
    CASE _InstanceState[E_INSTANCE.OUTFEED_ROBOT_R1].State
    OF
    E_INSTANCE_STATE.DISABLED:
      CASE _InstanceState[E_INSTANCE.OUTFEED_ROBOT_R1].Progress
      OF
      E_PROGRESS.PROGRESS_BUSY:
        IF (_ItfProcessCollector[E_INSTANCE.OUTFEED_ROBOT_R1].QueueProcessCount < 12)
        THEN
          _InstanceCtrl[E_INSTANCE.OUTFEED_ROBOT_R1].Cmd      := E_INSTANCE_CMD.DISABLE;
  
          IF NOT (_ItfProcessCollector[E_INSTANCE.OUTFEED_ROBOT_R1].GetBit(_wDisable, TO_BYTE(E_INSTANCE.OUTFEED_ROBOT_R1-1)))
          THEN
            _wDisable                                         := _ItfProcessCollector[E_INSTANCE.OUTFEED_ROBOT_R1].
                                                                 SetBit(_wDisable, TO_BYTE(E_INSTANCE.OUTFEED_ROBOT_R1-1));

            IF (_MessageLevel > E_MessageType.eMessageError)
            THEN
              _stMsg.eType                                    := E_MessageType.eMessageInfo;
              _stMsg.eSubdevice                               := e_Subdevice.Application_Finish;
              _stMsg.iErrorNumber                             := 0;
              _stMsg.sText                                    := concat(TO_STRING(E_INSTANCE.OUTFEED_ROBOT_R1), ': _wDisable ');
              _stMsg.sText                                    := concat(_stMsg.sText, _ItfProcessCollector[E_INSTANCE.OUTFEED_ROBOT_R1].BitsToString(_wDisable));
              f_MessageSet(_stMsg);
            END_IF
          END_IF
        ELSE
          _InstanceCtrl[E_INSTANCE.OUTFEED_ROBOT_R1].Cmd      := E_INSTANCE_CMD.ENABLE;
        END_IF
      END_CASE

      E_INSTANCE_STATE.ENABLED:
        CASE _InstanceState[E_INSTANCE.OUTFEED_ROBOT_R1].Progress
        OF
          E_PROGRESS.PROGRESS_OCCUPIED:
            _InstanceCtrl[E_INSTANCE.OUTFEED_ROBOT_R1].Cmd    := E_INSTANCE_CMD.PROCEED;
        END_CASE


      E_INSTANCE_STATE.WORKING:
        CASE _InstanceState[E_INSTANCE.OUTFEED_ROBOT_R1].Progress
        OF
          E_PROGRESS.PROGRESS_BUSY:
            _tonProcess [E_INSTANCE.OUTFEED_ROBOT_R1]
                                                  (IN         := FALSE, 
                                                   PT         := _tProcess[E_INSTANCE.OUTFEED_ROBOT_R1]);

            _InstanceCtrl[E_INSTANCE.OUTFEED_ROBOT_R1].Cmd    := E_INSTANCE_CMD.WORK;
    

          E_PROGRESS.PROGRESS_CHECK:
            _tonProcess [E_INSTANCE.OUTFEED_ROBOT_R1]
                                                  (IN         := TRUE, 
                                                   PT         := _tProcess[E_INSTANCE.OUTFEED_ROBOT_R1]);
    
            IF _tonProcess [E_INSTANCE.OUTFEED_ROBOT_R1].Q
            THEN
              _InstanceCtrl[E_INSTANCE.OUTFEED_ROBOT_R1].Cmd  := E_INSTANCE_CMD.FINISH;
            END_IF
        END_CASE

      E_INSTANCE_STATE.FINISH:
        CASE _InstanceState[E_INSTANCE.OUTFEED_ROBOT_R1].Progress
        OF
          E_PROGRESS.PROGRESS_BUSY:
            _InstanceCtrl[E_INSTANCE.OUTFEED_ROBOT_R1].Cmd    := E_INSTANCE_CMD.FINISH;

          E_PROGRESS.PROGRESS_DONE:
            _InstanceCtrl[E_INSTANCE.OUTFEED_ROBOT_R1].Cmd    := E_INSTANCE_CMD.DISABLE;
        END_CASE
      END_CASE

    //-------------------------------------------------------------------------
    // E_INSTANCE.OUTFEED_ROBOT_R2
    //-------------------------------------------------------------------------
    CASE _InstanceState[E_INSTANCE.OUTFEED_ROBOT_R2].State
    OF
    E_INSTANCE_STATE.DISABLED:
      CASE _InstanceState[E_INSTANCE.OUTFEED_ROBOT_R2].Progress
      OF
      E_PROGRESS.PROGRESS_BUSY:
        IF (_ItfProcessCollector[E_INSTANCE.OUTFEED_ROBOT_R2].QueueProcessCount < 12)
        THEN
          _InstanceCtrl[E_INSTANCE.OUTFEED_ROBOT_R2].Cmd      := E_INSTANCE_CMD.DISABLE;

          IF NOT (_ItfProcessCollector[E_INSTANCE.OUTFEED_ROBOT_R2].GetBit(_wDisable, TO_BYTE(E_INSTANCE.OUTFEED_ROBOT_R2-1)))
          THEN
            _wDisable                                         := _ItfProcessCollector[E_INSTANCE.OUTFEED_ROBOT_R2].
                                                                 SetBit(_wDisable, TO_BYTE(E_INSTANCE.OUTFEED_ROBOT_R2-1));

            IF (_MessageLevel > E_MessageType.eMessageError)
            THEN
              _stMsg.eType                                    := E_MessageType.eMessageInfo;
              _stMsg.eSubdevice                               := e_Subdevice.Application_Finish;
              _stMsg.iErrorNumber                             := 0;
              _stMsg.sText                                    := concat(TO_STRING(E_INSTANCE.OUTFEED_ROBOT_R2), ': _wDisable ');
              _stMsg.sText                                    := concat(_stMsg.sText, _ItfProcessCollector[E_INSTANCE.OUTFEED_ROBOT_R2].BitsToString(_wDisable));
              f_MessageSet(_stMsg);
            END_IF
          END_IF
        ELSE
          _InstanceCtrl[E_INSTANCE.OUTFEED_ROBOT_R2].Cmd      := E_INSTANCE_CMD.ENABLE;
        END_IF
      END_CASE

      E_INSTANCE_STATE.ENABLED:
        CASE _InstanceState[E_INSTANCE.OUTFEED_ROBOT_R2].Progress
        OF
          E_PROGRESS.PROGRESS_OCCUPIED:
            _InstanceCtrl[E_INSTANCE.OUTFEED_ROBOT_R2].Cmd    := E_INSTANCE_CMD.PROCEED;
        END_CASE

      E_INSTANCE_STATE.WORKING:
        CASE _InstanceState[E_INSTANCE.OUTFEED_ROBOT_R2].Progress
        OF
          E_PROGRESS.PROGRESS_BUSY:
            _tonProcess [E_INSTANCE.OUTFEED_ROBOT_R2]
                                                  (IN         := FALSE, 
                                                   PT         := _tProcess[E_INSTANCE.OUTFEED_ROBOT_R2]);

            _InstanceCtrl[E_INSTANCE.OUTFEED_ROBOT_R2].Cmd    := E_INSTANCE_CMD.WORK;

    
          E_PROGRESS.PROGRESS_CHECK:
            _tonProcess [E_INSTANCE.OUTFEED_ROBOT_R2]
                                                  (IN         := TRUE, 
                                                   PT         := _tProcess[E_INSTANCE.OUTFEED_ROBOT_R2]);
    
            IF _tonProcess [E_INSTANCE.OUTFEED_ROBOT_R2].Q
            THEN
              _InstanceCtrl[E_INSTANCE.OUTFEED_ROBOT_R2].Cmd  := E_INSTANCE_CMD.FINISH;
            END_IF
        END_CASE

      E_INSTANCE_STATE.FINISH:
        CASE _InstanceState[E_INSTANCE.OUTFEED_ROBOT_R2].Progress
        OF
          E_PROGRESS.PROGRESS_BUSY:
            _InstanceCtrl[E_INSTANCE.OUTFEED_ROBOT_R2].Cmd    := E_INSTANCE_CMD.FINISH;

          E_PROGRESS.PROGRESS_DONE:
            _InstanceCtrl[E_INSTANCE.OUTFEED_ROBOT_R2].Cmd    := E_INSTANCE_CMD.DISABLE;
        END_CASE
      END_CASE

    //-------------------------------------------------------------------------
    // E_INSTANCE.SENDER_FAST
    //-------------------------------------------------------------------------
    CASE _InstanceState[E_INSTANCE.SENDER_FAST].State
    OF
      E_INSTANCE_STATE.DISABLED:
        CASE _InstanceState[E_INSTANCE.SENDER_FAST].Progress
        OF
          E_PROGRESS.PROGRESS_BUSY:
            IF NOT (_ItfProcessCollector[E_INSTANCE.OUTFEED_ROBOT_R1].QueueProcessCount < 12) OR 
               NOT (_ItfProcessCollector[E_INSTANCE.OUTFEED_ROBOT_R2].QueueProcessCount < 12)
            THEN
              _InstanceCtrl[E_INSTANCE.SENDER_FAST].Cmd       := E_INSTANCE_CMD.ENABLE;

            ELSIF (_ItfProcessCollector[E_INSTANCE.SENDER_FAST].QueueProcessCount > 0)
            THEN
              _InstanceCtrl[E_INSTANCE.SENDER_FAST].Cmd       := E_INSTANCE_CMD.ENABLE;
            ELSE
              _InstanceCtrl[E_INSTANCE.SENDER_FAST].Cmd       := E_INSTANCE_CMD.DISABLE;

              IF NOT (_ItfProcessCollector[E_INSTANCE.SENDER_FAST].GetBit(_wDisable, TO_BYTE(E_INSTANCE.SENDER_FAST-1)))
              THEN
                _wDisable                                     := _ItfProcessCollector[E_INSTANCE.SENDER_FAST].
                                                                 SetBit(_wDisable, TO_BYTE(E_INSTANCE.SENDER_FAST-1));
    
                IF (_MessageLevel > E_MessageType.eMessageError)
                THEN
                  _stMsg.eType                                := E_MessageType.eMessageInfo;
                  _stMsg.eSubdevice                           := e_Subdevice.Application_Finish;
                  _stMsg.iErrorNumber                         := 0;
                  _stMsg.sText                                := concat(TO_STRING(E_INSTANCE.SENDER_FAST), ': _wDisable ');
                  _stMsg.sText                                := concat(_stMsg.sText, _ItfProcessCollector[E_INSTANCE.SENDER_FAST].BitsToString(_wDisable));
                  f_MessageSet(_stMsg);
                END_IF
              END_IF
            END_IF
        END_CASE

      E_INSTANCE_STATE.FINISH:
        CASE _InstanceState[E_INSTANCE.SENDER_FAST].Progress
        OF
          E_PROGRESS.PROGRESS_BUSY:
            _InstanceCtrl[E_INSTANCE.SENDER_FAST].Cmd         := E_INSTANCE_CMD.FINISH;
        END_CASE
      END_CASE
END_CASE
//-----------------------------------------------------------------------------
//-----------------------------------------------------------------------------
CASE _eState
OF
  E_PROGRESS.PROGRESS_STILL_WORKING:
    _XtsTransportCtrl.Cmd                                 := E_XTS_TRANSPORT_CTRL.CMD_GROUP_STOP;
  
    IF (_XtsTransportState.State = E_XTS_TRANSPORT_STATE.TRANSPORT_GROUP_STOP + E_PROGRESS.PROGRESS_ERROR)
    THEN
      _eState                                             := E_PROGRESS.PROGRESS_ERROR;

      _stMsg.eType                  := E_MessageType.eMessageError;
      _stMsg.eSubdevice             := e_Subdevice.Application_Finish;
      _stMsg.iErrorNumber           := 0;
      _stMsg.sText                  := concat(TO_STRING(_eState), ': ');
      f_MessageSet(_stMsg);

  
    ELSIF (_XtsTransportState.State = E_XTS_TRANSPORT_STATE.TRANSPORT_GROUP_STOP + E_PROGRESS.PROGRESS_DONE)
    THEN
      _eState                                             := E_PROGRESS.PROGRESS_DONE;

      IF (_MessageLevel > E_MessageType.eMessageError)
      THEN
        _stMsg.eType                := E_MessageType.eMessageInfo;
        _stMsg.eSubdevice           := e_Subdevice.Application_Finish;
        _stMsg.iErrorNumber         := 0;
        _stMsg.sText                := concat(TO_STRING(_eState), ': ');
        f_MessageSet(_stMsg);
      END_IF
    END_IF
END_CASE
//-----------------------------------------------------------------------------
//-----------------------------------------------------------------------------

Finish                            := _eState;
END_METHOD

METHOD Init       : E_PROGRESS // used only for first cycle startup, 
                               // use method Clear during operations if you have to clean up the instances 
VAR_INPUT
  Execute         : BOOL;
END_VAR
VAR_INST
  _nIdx,
  _nErrorId       : UDINT;
  _eState         : E_PROGRESS;
END_VAR
//-----------------------------------------------------------------------------
IF NOT Execute 
THEN 
	_eState                                         := E_PROGRESS.PROGRESS_INIT; 
END_IF 
//-----------------------------------------------------------------------------
IF NOT Check() 
THEN 
	Init                                            := E_PROGRESS.PROGRESS_ERROR; 
	RETURN; 
END_IF
//-----------------------------------------------------------------------------
//-----------------------------------------------------------------------------
CASE _eState
OF
  //---------------------------------------------------------------------------------------------------------------
  //---------------------------------------------------------------------------------------------------------------
  E_PROGRESS.PROGRESS_INIT:                   // startup procedure for your application
    IF Execute
    THEN
      _eState                                       := E_PROGRESS.PROGRESS_BUSY;

      IF (_MessageLevel > E_MessageType.eMessageError)
      THEN
        _stMsg.eType            := E_MessageType.eMessageInfo;
        _stMsg.eSubdevice       := e_Subdevice.Application_Init;
        _stMsg.iErrorNumber     := 0;
        _stMsg.sText            := concat(TO_STRING(_eState), ': ');
        f_MessageSet(_stMsg);
      END_IF

      IF (GVL_APPLICATION.bOutput_R1R2)
      THEN
        MAIN_APP.ProcessInit_R1R2();
      ELSE
        MAIN_APP.ProcessInit_CLAMP();
      END_IF

      FOR _nIdx := 1 TO MAX_PROCESS
      DO
        _InstanceCtrl[_nIdx].Cmd                    := E_INSTANCE_CMD.INIT;
      END_FOR
    END_IF
  //---------------------------------------------------------------------------------------------------------------
  //---------------------------------------------------------------------------------------------------------------
  E_PROGRESS.PROGRESS_BUSY:
    _InstanceCtrl[E_INSTANCE.BUFFER_INFEED].Cmd   := E_INSTANCE_CMD.DISABLE;
    //-----------------------------------------------------------------------------------
    CASE _InstanceState[E_INSTANCE.BUFFER_INFEED].State
    OF
      E_INSTANCE_STATE.DISABLED:
        CASE _InstanceState[E_INSTANCE.BUFFER_INFEED].Progress
        OF
          E_PROGRESS.PROGRESS_BUSY:           // check for startup to be done
            _eState                               := E_PROGRESS.PROGRESS_PREPARE; // go check next insatnce
        END_CASE
    END_CASE

  //---------------------------------------------------------------------------------------------------------------
  //---------------------------------------------------------------------------------------------------------------
  E_PROGRESS.PROGRESS_PREPARE:
    _InstanceCtrl[E_INSTANCE.INFEED].Cmd          := E_INSTANCE_CMD.DISABLE;
    //-----------------------------------------------------------------------------------
    CASE _InstanceState[E_INSTANCE.INFEED].State
    OF
      E_INSTANCE_STATE.DISABLED:
        CASE _InstanceState[E_INSTANCE.INFEED].Progress
        OF
          E_PROGRESS.PROGRESS_BUSY:           // check for startup to be done
          _eState                                 := E_PROGRESS.PROGRESS_STARTUP; // go check next insatnce
        END_CASE
    END_CASE

  //---------------------------------------------------------------------------------------------------------------
  //---------------------------------------------------------------------------------------------------------------
  E_PROGRESS.PROGRESS_STARTUP:
    _InstanceCtrl[E_INSTANCE.BUFFER_OUTFEED].Cmd   := E_INSTANCE_CMD.DISABLE;
    //-----------------------------------------------------------------------------------
    CASE _InstanceState[E_INSTANCE.BUFFER_OUTFEED].State
    OF
      E_INSTANCE_STATE.DISABLED:
        CASE _InstanceState[E_INSTANCE.BUFFER_OUTFEED].Progress
        OF
          E_PROGRESS.PROGRESS_BUSY:           // check for startup to be done
          _eState                                 := E_PROGRESS.PROGRESS_CHECK; // go check next insatnce
        END_CASE
    END_CASE

  //---------------------------------------------------------------------------------------------------------------
  //---------------------------------------------------------------------------------------------------------------
  E_PROGRESS.PROGRESS_CHECK:
    _InstanceCtrl[E_INSTANCE.OUTFEED_ROBOT_R1].Cmd   := E_INSTANCE_CMD.DISABLE;
    //-----------------------------------------------------------------------------------
    CASE _InstanceState[E_INSTANCE.OUTFEED_ROBOT_R1].State
    OF
      E_INSTANCE_STATE.DISABLED:
        CASE _InstanceState[E_INSTANCE.OUTFEED_ROBOT_R1].Progress
        OF
          E_PROGRESS.PROGRESS_BUSY:           // check for startup to be done
          _eState                                 := E_PROGRESS.PROGRESS_OCCUPIED; // go check next insatnce
        END_CASE
    END_CASE

  //---------------------------------------------------------------------------------------------------------------
  //---------------------------------------------------------------------------------------------------------------
  E_PROGRESS.PROGRESS_OCCUPIED:
    _InstanceCtrl[E_INSTANCE.OUTFEED_ROBOT_R2].Cmd   := E_INSTANCE_CMD.DISABLE;
    //-----------------------------------------------------------------------------------
    CASE _InstanceState[E_INSTANCE.OUTFEED_ROBOT_R2].State
    OF
      E_INSTANCE_STATE.DISABLED:
        CASE _InstanceState[E_INSTANCE.OUTFEED_ROBOT_R2].Progress
        OF
          E_PROGRESS.PROGRESS_BUSY:           // check for startup to be done
          _eState                                 := E_PROGRESS.PROGRESS_WORKING; // go check next insatnce
        END_CASE
    END_CASE

  //---------------------------------------------------------------------------------------------------------------
  //---------------------------------------------------------------------------------------------------------------
  E_PROGRESS.PROGRESS_WORKING:
    _InstanceCtrl[E_INSTANCE.SENDER_FAST].Cmd     := E_INSTANCE_CMD.DISABLE;
    //-----------------------------------------------------------------------------------
    CASE _InstanceState[E_INSTANCE.SENDER_FAST].State
    OF
      E_INSTANCE_STATE.DISABLED:
        CASE _InstanceState[E_INSTANCE.SENDER_FAST].Progress
        OF
          E_PROGRESS.PROGRESS_BUSY:           // check for startup to be done
          _eState                                 := E_PROGRESS.PROGRESS_STILL_WORKING; // go check next insatnce
        END_CASE
    END_CASE

  //---------------------------------------------------------------------------------------------------------------
  //---------------------------------------------------------------------------------------------------------------
  E_PROGRESS.PROGRESS_STILL_WORKING:
    _InstanceCtrl[E_INSTANCE.SENDER_BUFFER_INFEED].Cmd   := E_INSTANCE_CMD.DISABLE;
    //-----------------------------------------------------------------------------------
    CASE _InstanceState[E_INSTANCE.SENDER_BUFFER_INFEED].State
    OF
      E_INSTANCE_STATE.DISABLED:
        CASE _InstanceState[E_INSTANCE.SENDER_BUFFER_INFEED].Progress
        OF
          E_PROGRESS.PROGRESS_BUSY:           // check for startup to be done
          _eState                                 := E_PROGRESS.PROGRESS_DONE;
        END_CASE
    END_CASE
END_CASE
//-----------------------------------------------------------------------------
//-----------------------------------------------------------------------------

Init                                              := _eState;
END_METHOD

PROPERTY InstanceCtrl : REFERENCE TO ARRAY[1..MAX_PROCESS] OF ST_INSTANCE_CTRL
SET
_InstanceCtrl REF= InstanceCtrl;
END_SET
END_PROPERTY

PROPERTY InstanceState : REFERENCE TO ARRAY[1..MAX_PROCESS] OF ST_INSTANCE_STATE
SET
_InstanceState REF= InstanceState;
END_SET
END_PROPERTY

METHOD ListData   : E_PROGRESS  // simulates data entry from transfersystem into BUFFER_INFEED linked list
VAR_INPUT
  Start           : BOOL;
  Reset           : BOOL;
END_VAR
VAR_INST
  _nBit,
  _nExp           : BYTE;
  _nMod           : UINT := 5;
  _nCount         : UINT;
  _eStateProgress : E_PROGRESS;

  _ProcessData    : ST_PROCESS_DATA;
  _Rslt           : ST_PROCESS_LIST_RESULT;

  _nMinListCount  : UDINT := 1;
  _nWaitcountLast,
  _nWaitCount     : UDINT;

  _tMsg           : ST_Message;
  _eMessageLevel  : E_MessageType;  // manual local switch for enabling info messages
END_VAR
IF Reset
THEN
  _nCount                     := 1;
  _eStateProgress             := E_PROGRESS.PROGRESS_INIT;
  _ItfProcessList[E_INSTANCE.BUFFER_INFEED].InitList();
END_IF

_tMsg.eDevice                 := _stMsg.eDevice; 

CASE _eStateProgress
OF
   E_PROGRESS.PROGRESS_INIT:
    IF Start
    THEN
      _eStateProgress         :=  E_PROGRESS.PROGRESS_BUSY;
    END_IF

  E_PROGRESS.PROGRESS_BUSY:
    CASE _nLoadCase
    OF
      0:  // fully loaded
        _eStateProgress       := E_PROGRESS.PROGRESS_CHECK;
        _nLoadCaseOld         := _nLoadCase;

        IF (_eMessageLevel > E_MessageType.eMessageError)
        THEN
          _tMsg.eType          := E_MessageType.eMessageInfo;
          _tMsg.eSubdevice     := e_Subdevice.Application;
          _tMsg.iErrorNumber   := _nLoadCase;
          _tMsg.sText          := concat(TO_STRING(_eState), ': ListData');
          f_MessageSet(_stMsg);
        END_IF


      1:  // static bits
        _eStateProgress       := E_PROGRESS.PROGRESS_PREPARE;
        _nLoadCaseOld         := _nLoadCase;

        IF (_eMessageLevel > E_MessageType.eMessageError)
        THEN
          _tMsg.eType          := E_MessageType.eMessageInfo;
          _tMsg.eSubdevice     := e_Subdevice.Application;
          _tMsg.iErrorNumber   := _nLoadCase;
          _tMsg.sText          := concat(TO_STRING(_eState), ': ListData');
          f_MessageSet(_stMsg);
        END_IF


      2:  // incrementing bits
        _eStateProgress       := E_PROGRESS.PROGRESS_STARTUP;
        _nLoadCaseOld         := _nLoadCase;

        IF (_eMessageLevel > E_MessageType.eMessageError)
        THEN
          _tMsg.eType          := E_MessageType.eMessageInfo;
          _tMsg.eSubdevice     := e_Subdevice.Application;
          _tMsg.iErrorNumber   := _nLoadCase;
          _tMsg.sText          := concat(TO_STRING(_eState), ': ListData');
          f_MessageSet(_stMsg);
        END_IF


      99:
        _eStateProgress       := E_PROGRESS.PROGRESS_WORKING;
        _ProcessData.wTarget  := 0;

        IF (_eMessageLevel > E_MessageType.eMessageError)
        THEN
          _tMsg.eType          := E_MessageType.eMessageInfo;
          _tMsg.eSubdevice     := e_Subdevice.Application;
          _tMsg.iErrorNumber   := _nLoadCase;
          _tMsg.sText          := concat(TO_STRING(_eState), ': _ProcessData.wTarget: ');
          _tMsg.sText          := concat(_stMsg.sText, _ItfProcessCollector[E_INSTANCE.BUFFER_INFEED].BitsToString(_ProcessData.wTarget));
          f_MessageSet(_stMsg);
        END_IF
        _nLoadCase            := _nLoadCaseOld;

    ELSE
        _eStateProgress       := E_PROGRESS.PROGRESS_STARTUP;
    END_CASE
    _nWaitCount               := 0; 
END_CASE
CASE _eStateProgress
OF
  E_PROGRESS.PROGRESS_PREPARE:
    _eStateProgress           := E_PROGRESS.PROGRESS_WORKING;
    _nExp                     := TO_BYTE(ItfProcessCollector[E_INSTANCE.INFEED].StationCount);
    _ProcessData.wTarget      := _ItfProcessCollector[E_INSTANCE.BUFFER_INFEED].To_T_Process(_nExp);

    IF (_nCount MOD _nMod = 0)
    THEN
      _nBit                   := SEL((_nBit>_nExp), _nBit+1, 0);
      _ProcessData.wTarget    := _ItfProcessCollector[E_INSTANCE.BUFFER_INFEED].DelBit(_ProcessData.wTarget, _nBit);
    END_IF
    IF (_nCount MOD (8) = 0)
    THEN
      _nBit                   := 1;
      _ProcessData.wTarget    := _ItfProcessCollector[E_INSTANCE.BUFFER_INFEED].DelBit(_ProcessData.wTarget, _nBit);
    END_IF
    IF (_nCount MOD (16) = 0)
    THEN
      _nBit                   := 2;
      _ProcessData.wTarget    := _ItfProcessCollector[E_INSTANCE.BUFFER_INFEED].DelBit(_ProcessData.wTarget, _nBit);
    END_IF
    IF (_nCount MOD (24) = 0)
    THEN
      _nBit                   := 3;
      _ProcessData.wTarget    := _ItfProcessCollector[E_INSTANCE.BUFFER_INFEED].DelBit(_ProcessData.wTarget, _nBit);
    END_IF
    IF (_nCount MOD (32) = 0)
    THEN
      _nBit                   := 4;
      _ProcessData.wTarget    := _ItfProcessCollector[E_INSTANCE.BUFFER_INFEED].DelBit(_ProcessData.wTarget, _nBit);
    END_IF
    IF (_nCount MOD (40) = 0)
    THEN
      _nBit                   := 5;
      _ProcessData.wTarget    := _ItfProcessCollector[E_INSTANCE.BUFFER_INFEED].DelBit(_ProcessData.wTarget, _nBit);
    END_IF
    IF (_nCount MOD (48) = 0)
    THEN
      _nBit                   := 6;
      _ProcessData.wTarget    := _ItfProcessCollector[E_INSTANCE.BUFFER_INFEED].DelBit(_ProcessData.wTarget, _nBit);
    END_IF
    IF (_nCount MOD (60) = 0)
    THEN
      _nBit                   := 7;
      _ProcessData.wTarget    := _ItfProcessCollector[E_INSTANCE.BUFFER_INFEED].DelBit(_ProcessData.wTarget, _nBit);
    END_IF
    IF (_nCount MOD (72) = 0)
    THEN
      _nBit                   := 8;
      _ProcessData.wTarget    := _ItfProcessCollector[E_INSTANCE.BUFFER_INFEED].DelBit(_ProcessData.wTarget, _nBit);
    END_IF
    IF (_nCount MOD (84) = 0)
    THEN
      _nBit                   := 9;
      _ProcessData.wTarget    := _ItfProcessCollector[E_INSTANCE.BUFFER_INFEED].DelBit(_ProcessData.wTarget, _nBit);
    END_IF
    IF (_nCount MOD (96) = 0)
    THEN
      _nBit                   := 10;
      _ProcessData.wTarget    := _ItfProcessCollector[E_INSTANCE.BUFFER_INFEED].DelBit(_ProcessData.wTarget, _nBit);
    END_IF
    IF (_nCount MOD (108) = 0)
    THEN
      _nBit                   := 11;
      _ProcessData.wTarget    := _ItfProcessCollector[E_INSTANCE.BUFFER_INFEED].DelBit(_ProcessData.wTarget, _nBit);
    END_IF
END_CASE
CASE _eStateProgress
OF
  E_PROGRESS.PROGRESS_STARTUP:
    _eStateProgress           := E_PROGRESS.PROGRESS_WORKING;
    _nExp                     := TO_BYTE(ItfProcessCollector[E_INSTANCE.INFEED].StationCount);
    _ProcessData.wTarget      := _ItfProcessCollector[E_INSTANCE.BUFFER_INFEED].To_T_Process(_nExp);

    IF (_nCount MOD _nMod = 0)
    THEN
      _nBit                   := SEL((_nBit>_nExp), _nBit+1, 0);
      _ProcessData.wTarget    := _ItfProcessCollector[E_INSTANCE.BUFFER_INFEED].DelBit(_ProcessData.wTarget, _nBit);
    END_IF
(*
    IF (_nCount MOD (8) = 0)
    THEN
      _nBit                   := SEL((_nBit>_nExp), _nBit+1, 0);
      _ProcessData.wTarget    := _ItfProcessCollector[E_INSTANCE.BUFFER_INFEED].DelBit(_ProcessData.wTarget, _nBit);
    END_IF
    IF (_nCount MOD (16) = 0)
    THEN
      _nBit                   := SEL((_nBit>_nExp), _nBit+1, 0);
      _ProcessData.wTarget    := _ItfProcessCollector[E_INSTANCE.BUFFER_INFEED].DelBit(_ProcessData.wTarget, _nBit);
    END_IF
    IF (_nCount MOD (24) = 0)
    THEN
      _nBit                   := SEL((_nBit>_nExp), _nBit+1, 0);
      _ProcessData.wTarget    := _ItfProcessCollector[E_INSTANCE.BUFFER_INFEED].DelBit(_ProcessData.wTarget, _nBit);
    END_IF
    IF (_nCount MOD (32) = 0)
    THEN
      _nBit                   := SEL((_nBit>_nExp), _nBit+1, 0);
      _ProcessData.wTarget    := _ItfProcessCollector[E_INSTANCE.BUFFER_INFEED].DelBit(_ProcessData.wTarget, _nBit);
    END_IF
    IF (_nCount MOD (40) = 0)
    THEN
      _nBit                   := SEL((_nBit>_nExp), _nBit+1, 0);
      _ProcessData.wTarget    := _ItfProcessCollector[E_INSTANCE.BUFFER_INFEED].DelBit(_ProcessData.wTarget, _nBit);
    END_IF
    IF (_nCount MOD (48) = 0)
    THEN
      _nBit                   := SEL((_nBit>_nExp), _nBit+1, 0);
      _ProcessData.wTarget    := _ItfProcessCollector[E_INSTANCE.BUFFER_INFEED].DelBit(_ProcessData.wTarget, _nBit);
    END_IF
*)
END_CASE
CASE _eStateProgress
OF
  E_PROGRESS.PROGRESS_CHECK:
    _eStateProgress           := E_PROGRESS.PROGRESS_WORKING;
    _nExp                     := TO_BYTE(ItfProcessCollector[E_INSTANCE.INFEED].StationCount);
    _ProcessData.wTarget      := _ItfProcessCollector[E_INSTANCE.BUFFER_INFEED].To_T_Process(_nExp);

    IF (_eMessageLevel > E_MessageType.eMessageError)
    THEN
      _tMsg.eType            := E_MessageType.eMessageInfo;
      _tMsg.eSubdevice       := e_Subdevice.Application;
      _tMsg.iErrorNumber     := _nLoadCase;
      _tMsg.sText            := concat(TO_STRING(_eState), ': _ProcessData.wTarget: ');
      _tMsg.sText            := concat(_stMsg.sText, _ItfProcessCollector[E_INSTANCE.BUFFER_INFEED].BitsToString(_ProcessData.wTarget));
      f_MessageSet(_stMsg);
    END_IF
END_CASE
CASE _eStateProgress
OF
  E_PROGRESS.PROGRESS_WORKING:
    _Rslt                     := _ItfProcessList[E_INSTANCE.BUFFER_INFEED].AddTailValue(_ProcessData);

    IF (_Rslt.wState = 0)
    THEN
      _nCount                 := _nCount + 1;
      _eStateProgress         := E_PROGRESS.PROGRESS_OCCUPIED;
    ELSE
      _eStateProgress         := E_PROGRESS.PROGRESS_ERROR;
    END_IF
END_CASE
CASE _eStateProgress
OF
  E_PROGRESS.PROGRESS_OCCUPIED:
    _nWaitCount               := _nWaitCount + 1;

    IF (_ItfProcessList[E_INSTANCE.BUFFER_INFEED].Count < _nMinListCount)
    THEN
      _nWaitCountLast         := _nWaitCount;
      _eStateProgress         :=  E_PROGRESS.PROGRESS_INIT;
    END_IF
END_CASE

ListData                      := _eStateProgress;
END_METHOD

PROPERTY MessageLevel : e_MessageType
GET
MessageLevel := _MessageLevel;
END_GET
SET
_MessageLevel := MessageLevel;
END_SET
END_PROPERTY

METHOD Proceed : E_PROGRESS
VAR_INPUT
  Execute     : BOOL;
END_VAR
VAR_INST
  _nErrorId               : UDINT;
  _eState                 : E_PROGRESS;

  _nExp                   : BYTE;
  _WriteData              : ST_PROCESS_DATA;
  _WriteResult            : ST_PROCESS_LIST_RESULT;

  _eInst                  : E_INSTANCE;
  _TransportState         : E_XTS_TRANSPORT_STATE;
  _bDbg : BOOL;
END_VAR
//-----------------------------------------------------------------------------
IF NOT Execute 
THEN 
	_eState                       := E_PROGRESS.PROGRESS_INIT; 
END_IF 
//-----------------------------------------------------------------------------
IF NOT Check() 
THEN 
	Proceed                       := E_PROGRESS.PROGRESS_ERROR; 
	RETURN; 
END_IF
//-----------------------------------------------------------------------------
//-----------------------------------------------------------------------------
CASE _eState
OF
  E_PROGRESS.PROGRESS_INIT:
    IF Execute
    THEN
      _nErrorId                 := 0;

      IF (_XtsTransportState.GroupInfo.AxisCountEnabled = MAX_MOVER) AND
         (_XtsTransportState.GroupInfo.AxisCount        = MAX_MOVER)
      THEN
        _eState                 := E_PROGRESS.PROGRESS_BUSY;
        _XtsTransportCtrl.Cmd   := E_XTS_TRANSPORT_CTRL.CMD_NULL;

        IF (_MessageLevel > E_MessageType.eMessageError)
        THEN
          _stMsg.eType          := E_MessageType.eMessageInfo;
          _stMsg.eSubdevice     := e_Subdevice.Application_Proceed;
          _stMsg.iErrorNumber   := 0;
          _stMsg.sText          := concat(TO_STRING(_eState), ': ');
          f_MessageSet(_stMsg);
        END_IF
      ELSE
        _nErrorId               := _eState;

        _eState                 := E_PROGRESS.PROGRESS_ERROR;

        _stMsg.eType            := E_MessageType.eMessageError;
        _stMsg.eSubdevice       := e_Subdevice.Application_Proceed;
        _stMsg.iErrorNumber     := _nErrorId;
        _stMsg.sText            := concat(TO_STRING(_eState), ': ');
        _stMsg.sText            := concat(_stMsg.sText, TO_STRING(_XtsTransportState.GroupInfo.AxisCountEnabled));
        _stMsg.sText            := concat(_stMsg.sText, ' / ');
        _stMsg.sText            := concat(_stMsg.sText, TO_STRING(_XtsTransportState.GroupInfo.AxisCount));
        _stMsg.sText            := concat(_stMsg.sText, ' CaGroup Axis mismatch');
        f_MessageSet(_stMsg);
      END_IF
    END_IF


  E_PROGRESS.PROGRESS_BUSY:
    _XtsTransportCtrl.Cmd       := E_XTS_TRANSPORT_CTRL.CMD_TRANSPORT_RESTART;

    IF (_XtsTransportState.State = E_XTS_TRANSPORT_STATE.TRANSPORT_RESTART + E_PROGRESS.PROGRESS_ERROR)
    THEN
      _eState                   := E_PROGRESS.PROGRESS_ERROR;
      _TransportState           := _XtsTransportState.State MOD E_PROGRESS.PROGRESS_ERROR;

      _stMsg.eType              := E_MessageType.eMessageError;
      _stMsg.eSubdevice         := e_Subdevice.Application_Proceed;
      _stMsg.iErrorNumber       := _nErrorId;
      _stMsg.sText              := concat(TO_STRING(_eState), ': ');
      _stMsg.sText              := concat(_stMsg.sText, TO_STRING(_TransportState));
      f_MessageSet(_stMsg);

    ELSIF (_XtsTransportState.State = E_XTS_TRANSPORT_STATE.TRANSPORT_RESTART + E_PROGRESS.PROGRESS_DONE)
    THEN
      _eState                   := E_PROGRESS.PROGRESS_WORKING;
      _TransportState           := _XtsTransportState.State MOD E_PROGRESS.PROGRESS_DONE;

      IF (_MessageLevel > E_MessageType.eMessageError)
      THEN
        _stMsg.eType            := E_MessageType.eMessageInfo;
        _stMsg.eSubdevice       := e_Subdevice.Application_Proceed;
        _stMsg.iErrorNumber     := 0;
        _stMsg.sText            := concat(TO_STRING(_eState), ': ');
        _stMsg.sText            := concat(_stMsg.sText, TO_STRING(_TransportState));
        f_MessageSet(_stMsg);
      END_IF
    END_IF

END_CASE
//-----------------------------------------------------------------------------
//-----------------------------------------------------------------------------
CASE _eState
OF
  E_PROGRESS.PROGRESS_WORKING:
    ListData(TRUE, FALSE);    // start writing linked list entries into BUFFER_INFEED

    FOR _eInst := E_INSTANCE.BUFFER_INFEED TO E_INSTANCE.SENDER_BUFFER_INFEED
    DO
      // handshakes to instances: 
      // - deconstruct this for your own implementation
      CASE _InstanceState[_eInst].State
      OF
        E_INSTANCE_STATE.DISABLED:
          CASE _InstanceState[_eInst].Progress
          OF
            E_PROGRESS.PROGRESS_BUSY:
              _InstanceCtrl[_eInst].Cmd    := E_INSTANCE_CMD.ENABLE;
          END_CASE
      
        E_INSTANCE_STATE.ENABLED:
          CASE _InstanceState[_eInst].Progress
          OF
            E_PROGRESS.PROGRESS_OCCUPIED:
              _InstanceCtrl[_eInst].Cmd    := E_INSTANCE_CMD.PROCEED;
          END_CASE
      
        E_INSTANCE_STATE.WORKING:
          CASE _InstanceState[_eInst].Progress
          OF
            E_PROGRESS.PROGRESS_BUSY:
              _tonProcess [_eInst]
                              (IN         := FALSE, 
                               PT         := _tProcess[_eInst]);

              IF (_eInst > E_INSTANCE.OUTFEED_ROBOT_R2) OR
                 (_eInst < E_INSTANCE.OUTFEED_ROBOT_R1) OR
                 (_bSingleOutput) OR
                 NOT (GVL_APPLICATION.bOutput_R1R2)
              THEN
                _InstanceCtrl[_eInst].Cmd   := E_INSTANCE_CMD.WORK;
              ELSE
                IF (_InstanceState[E_INSTANCE.OUTFEED_ROBOT_R1].State = 
                    _InstanceState[E_INSTANCE.OUTFEED_ROBOT_R2].State )
                THEN
                  // in this example the outfeed instances are working in sync
                  _InstanceCtrl[_eInst].Cmd := E_INSTANCE_CMD.WORK;
                ELSE
                  CASE _InstanceState[E_INSTANCE.OUTFEED_ROBOT_R2].State
                  OF
                    E_INSTANCE_STATE.ENABLED:
                      // in case R2 is empty --> unload R1
                      _InstanceCtrl[E_INSTANCE.OUTFEED_ROBOT_R1].Cmd := E_INSTANCE_CMD.WORK;
                  END_CASE
                END_IF
              END_IF
      
      
            E_PROGRESS.PROGRESS_CHECK:
              _tonProcess [_eInst]
                              (IN         := TRUE, 
                               PT         := _tProcess[_eInst]);
      
              IF _tonProcess [_eInst].Q
              THEN
                _InstanceCtrl[_eInst].Cmd := E_INSTANCE_CMD.FINISH;
              END_IF
          END_CASE


        E_INSTANCE_STATE.FINISH:
          CASE _InstanceState[_eInst].Progress
          OF
            E_PROGRESS.PROGRESS_BUSY:
              _InstanceCtrl[_eInst].Cmd    := E_INSTANCE_CMD.FINISH;

            E_PROGRESS.PROGRESS_OCCUPIED:
              _InstanceCtrl[_eInst].Cmd    := E_INSTANCE_CMD.PROCEED;
          END_CASE
        END_CASE
    END_FOR
END_CASE
//-----------------------------------------------------------------------------
//-----------------------------------------------------------------------------

Proceed                            := _eState;
END_METHOD

PROPERTY ProcessLinkedLists : REFERENCE TO ARRAY[1..MAX_PROCESS] OF I_Process_LinkedList
SET
_ItfProcessList REF= ProcessLinkedLists;
END_SET
END_PROPERTY

PROPERTY State : REFERENCE TO ST_APP_STATE
SET
_State ref= State;
END_SET
END_PROPERTY

METHOD Work : E_PROGRESS  // cyclic handshakes with timers, 
                          // this procedure you have to build for your own application. 
                          // This simulated work method is here 
                          // because it was convinient for me to do so
VAR_INPUT
  Execute                 : BOOL;
END_VAR
VAR_INST
  _nErrorId               : UDINT;
  _eRslt,
  _eState                 : E_PROGRESS;

  _nExp                   : BYTE;
  _WriteData              : ST_PROCESS_DATA;
  _WriteResult            : ST_PROCESS_LIST_RESULT;

  _eInst                  : E_INSTANCE;
  _bDbg : BOOL;

  _TransportState         : E_XTS_TRANSPORT_STATE;
  _JobResult              : E_PROGRESS;
END_VAR
//-----------------------------------------------------------------------------
IF NOT Execute 
THEN 
	_eState                       := E_PROGRESS.PROGRESS_INIT; 
END_IF 
//-----------------------------------------------------------------------------
IF NOT Check() 
THEN 
	Work                          := E_PROGRESS.PROGRESS_ERROR; 
	RETURN; 
END_IF
//-----------------------------------------------------------------------------
//-----------------------------------------------------------------------------
CASE _eState
OF
  E_PROGRESS.PROGRESS_INIT:
    IF Execute
    THEN
      _nErrorId                 := 0;

      IF (_XtsTransportState.GroupInfo.AxisCountEnabled = MAX_MOVER) AND
         (_XtsTransportState.GroupInfo.AxisCount        = MAX_MOVER)
      THEN
        _eState                 := E_PROGRESS.PROGRESS_BUSY;
        _XtsTransportCtrl.Cmd   := E_XTS_TRANSPORT_CTRL.CMD_NULL;
        _eRslt                  := Clear(FALSE);

        IF (_MessageLevel > E_MessageType.eMessageError)
        THEN
          _stMsg.eType          := E_MessageType.eMessageInfo;
          _stMsg.eSubdevice     := e_Subdevice.Application_Work;
          _stMsg.iErrorNumber   := 0;
          _stMsg.sText          := concat(TO_STRING(_eState), ': ');
          f_MessageSet(_stMsg);
        END_IF
      ELSE
        _nErrorId               := _XtsTransportState.GroupInfo.AxisCountEnabled;
        _eState                 := E_PROGRESS.PROGRESS_ERROR;

        _stMsg.eType            := E_MessageType.eMessageError;
        _stMsg.eSubdevice       := e_Subdevice.Application_Work;
        _stMsg.iErrorNumber     := _nErrorId;
        _stMsg.sText            := concat(TO_STRING(_eState), ': ');
        _stMsg.sText            := concat(_stMsg.sText, TO_STRING(_XtsTransportState.GroupInfo.AxisCountEnabled));
        _stMsg.sText            := concat(_stMsg.sText, ' / ');
        _stMsg.sText            := concat(_stMsg.sText, TO_STRING(_XtsTransportState.GroupInfo.AxisCount));
        _stMsg.sText            := concat(_stMsg.sText, ' CaGroup Axis mismatch');
        f_MessageSet(_stMsg);
      END_IF
    END_IF


  E_PROGRESS.PROGRESS_BUSY:
    _eRslt                      := Clear(TRUE);

    IF (_eRslt = E_PROGRESS.PROGRESS_DONE)
    THEN
      _XtsTransportCtrl.Cmd     := E_XTS_TRANSPORT_CTRL.CMD_TRANSPORT_START;
  
      IF (_XtsTransportState.State = E_XTS_TRANSPORT_STATE.TRANSPORT_START + E_PROGRESS.PROGRESS_ERROR)
      THEN
        _eState                 := E_PROGRESS.PROGRESS_ERROR;
        _TransportState         := _XtsTransportState.State MOD E_PROGRESS.PROGRESS_ERROR;

        _stMsg.eType            := E_MessageType.eMessageError;
        _stMsg.eSubdevice       := e_Subdevice.Application_Work;
        _stMsg.iErrorNumber     := _nErrorId;
        _stMsg.sText            := concat(TO_STRING(_eState), ': ');
        _stMsg.sText            := concat(_stMsg.sText, TO_STRING(_TransportState));
        f_MessageSet(_stMsg);
  
      ELSIF (_XtsTransportState.State = E_XTS_TRANSPORT_STATE.TRANSPORT_START + E_PROGRESS.PROGRESS_DONE)
      THEN
        _eState                 := E_PROGRESS.PROGRESS_PREPARE;
        _TransportState         := _XtsTransportState.State MOD E_PROGRESS.PROGRESS_DONE;

        IF (_MessageLevel > E_MessageType.eMessageError)
        THEN
          _stMsg.eType          := E_MessageType.eMessageInfo;
          _stMsg.eSubdevice     := e_Subdevice.Application_Work;
          _stMsg.iErrorNumber   := 0;
          _stMsg.sText          := concat(TO_STRING(_eState), ': ');
          _stMsg.sText          := concat(_stMsg.sText, TO_STRING(_TransportState));
          f_MessageSet(_stMsg);
        END_IF
      END_IF
    END_IF
END_CASE
//-----------------------------------------------------------------------------
//-----------------------------------------------------------------------------
CASE _eState
OF
  E_PROGRESS.PROGRESS_PREPARE:  // SENDER_BUFFER_INFEED sends the first batch of movers to BUFFER_INFEED
                                //  - after sending the first batch 
                                //    --> the transfersystem (ListData) may start writing entries into BUFFER_INFEED
    CASE _InstanceState[E_INSTANCE.SENDER_BUFFER_INFEED].State
    OF
    E_INSTANCE_STATE.DISABLED:

      CASE _InstanceState[E_INSTANCE.SENDER_BUFFER_INFEED].Progress
      OF
      E_PROGRESS.PROGRESS_BUSY:
        _nExp                   := TO_BYTE(ItfProcessCollector[E_INSTANCE.INFEED].StationCount);
        _WriteData.wTarget      := _ItfProcessCollector[E_INSTANCE.SENDER_BUFFER_INFEED].To_T_Process(_nExp);

        _WriteResult            := _ItfProcessList[E_INSTANCE.SENDER_BUFFER_INFEED].AddTailValue(_WriteData);

        IF (_WriteResult.wState <> 0)
        THEN
          _eState               := E_PROGRESS.PROGRESS_ERROR;

          _stMsg.eType          := E_MessageType.eMessageError;
          _stMsg.eSubdevice     := e_Subdevice.Application_Work;
          _stMsg.iErrorNumber   := _WriteResult.wState;
          _stMsg.sText          := concat(TO_STRING(_eState), ': ');
          _stMsg.sText          := concat(_stMsg.sText, TO_STRING(e_Subdevice.Process_LinkedList_AddTail));
          f_MessageSet(_stMsg);

        ELSE
          ListData(FALSE, TRUE);    // init linked list from simulated transfersystem (timer based entry into linked list)
          _eState               := E_PROGRESS.PROGRESS_CHECK;

          IF (_MessageLevel > E_MessageType.eMessageError)
          THEN
            _stMsg.eType        := E_MessageType.eMessageInfo;
            _stMsg.eSubdevice   := e_Subdevice.Application_Work;
            _stMsg.iErrorNumber := 0;
            _stMsg.sText        := concat(TO_STRING(_eState), ': ');
            _stMsg.sText        := concat(_stMsg.sText, TO_STRING(e_Subdevice.Process_LinkedList_AddTail));
            f_MessageSet(_stMsg);
          END_IF
        END_IF
      END_CASE
    END_CASE
END_CASE
//-----------------------------------------------------------------------------
//-----------------------------------------------------------------------------
CASE _eState
OF
  E_PROGRESS.PROGRESS_CHECK:
    _eState := E_PROGRESS.PROGRESS_OCCUPIED; 
END_CASE
//-----------------------------------------------------------------------------
//-----------------------------------------------------------------------------
CASE _eState
OF
  E_PROGRESS.PROGRESS_OCCUPIED:
    _eState := E_PROGRESS.PROGRESS_WORKING;

    IF (_MessageLevel > E_MessageType.eMessageError)
    THEN
      _stMsg.eType            := E_MessageType.eMessageInfo;
      _stMsg.eSubdevice       := e_Subdevice.Application_Work;
      _stMsg.iErrorNumber     := 0;
      _stMsg.sText            := concat(TO_STRING(_eState), ': ');
      f_MessageSet(_stMsg);
    END_IF
END_CASE
//-----------------------------------------------------------------------------
//-----------------------------------------------------------------------------
CASE _eState
OF
  E_PROGRESS.PROGRESS_WORKING:
    ListData(TRUE, FALSE);    // start writing linked list entries into BUFFER_INFEED

    FOR _eInst := E_INSTANCE.BUFFER_INFEED TO E_INSTANCE.SENDER_BUFFER_INFEED
    DO
      // handshakes to instances: 
      // - deconstruct this for your own implementation
      CASE _InstanceState[_eInst].State
      OF
        E_INSTANCE_STATE.DISABLED:
          CASE _InstanceState[_eInst].Progress
          OF
            E_PROGRESS.PROGRESS_BUSY:
              _InstanceCtrl[_eInst].Cmd    := E_INSTANCE_CMD.ENABLE;
          END_CASE
      
        E_INSTANCE_STATE.ENABLED:
          CASE _InstanceState[_eInst].Progress
          OF
            E_PROGRESS.PROGRESS_OCCUPIED:
              _InstanceCtrl[_eInst].Cmd    := E_INSTANCE_CMD.PROCEED;
          END_CASE

        E_INSTANCE_STATE.WORKING:
          CASE _InstanceState[_eInst].Progress
          OF
            E_PROGRESS.PROGRESS_BUSY:
              _tonProcess [_eInst]
                              (IN         := FALSE, 
                               PT         := _tProcess[_eInst]);


              IF (_eInst > E_INSTANCE.OUTFEED_ROBOT_R2) OR
                 (_eInst < E_INSTANCE.OUTFEED_ROBOT_R1) OR
                 (_bSingleOutput) OR
                 NOT (GVL_APPLICATION.bOutput_R1R2)
              THEN
                _InstanceCtrl[_eInst].Cmd   := E_INSTANCE_CMD.WORK;
              ELSE
                IF (_InstanceState[E_INSTANCE.OUTFEED_ROBOT_R1].State = 
                    _InstanceState[E_INSTANCE.OUTFEED_ROBOT_R2].State )
                THEN
                  // in this example the outfeed instances are working in sync
                  _InstanceCtrl[_eInst].Cmd := E_INSTANCE_CMD.WORK;
                END_IF
              END_IF
      
      
            E_PROGRESS.PROGRESS_CHECK:
              _tonProcess [_eInst]
                              (IN         := TRUE, 
                               PT         := _tProcess[_eInst]);
      
              IF _tonProcess [_eInst].Q
              THEN
                _InstanceCtrl[_eInst].Cmd := E_INSTANCE_CMD.FINISH;
              END_IF
          END_CASE


        E_INSTANCE_STATE.FINISH:
          CASE _InstanceState[_eInst].Progress
          OF
            E_PROGRESS.PROGRESS_BUSY:
              _tonProcess [_eInst]
                              (IN         := FALSE, 
                               PT         := _tProcess[_eInst]);

              _InstanceCtrl[_eInst].Cmd    := E_INSTANCE_CMD.FINISH;

            E_PROGRESS.PROGRESS_OCCUPIED:
              _InstanceCtrl[_eInst].Cmd    := E_INSTANCE_CMD.PROCEED;
          END_CASE
        END_CASE
    END_FOR
END_CASE
//-----------------------------------------------------------------------------
//-----------------------------------------------------------------------------

Work                            := _eState;
END_METHOD

PROPERTY WriteTimeVariant : bool
GET
WriteTimeVariant := _bWriteTimeVariant;
END_GET
SET
_bWriteTimeVariant := WriteTimeVariant;
END_SET
END_PROPERTY

PROPERTY XtsTransportCtrl : REFERENCE TO ST_XTS_TRANSPORT_CTRL
SET
_XtsTransportCtrl REF= XtsTransportCtrl;
END_SET
END_PROPERTY

PROPERTY XtsTransportState : REFERENCE TO ST_XTS_TRANSPORT_STATE
SET
_XtsTransportState REF= XtsTransportState;
END_SET
END_PROPERTY

END_FUNCTION_BLOCK

(* stored: Version 1.1.0.1, ProductVersion 3.1.4026.12
   POU fb_Application: Id {2a567699-b424-4e74-9f05-5574e5bc55b4}, SpecialFunc None
   Folder methods: Id {c1859e40-d269-4bfd-b7e9-641110aadb02}
   Folder properties: Id {440d7726-2a35-48b4-b212-3894cea03b12}
   Method Check: Id {b52b527b-139a-44b4-ab60-3e8b71488a0f}
   Method Clear: Id {a3ccc2ba-024d-44f1-adda-ac1f1be496a7}
   Method Cmd: Id {5496702b-60b7-475b-bef7-df563de1292d}
   Property CollectorInterface: Id {098e7272-6200-4a40-80ef-8c196e915eab}
   Set Set: Id {895034ec-84e5-4403-8b5f-9feedb87d7e4}
   Property Ctrl: Id {046d33ef-169b-4a2a-8c66-b97cf29ea596}
   Set Set: Id {a97b0d64-fc43-43a2-a267-33d710f4a902}
   Method Disable: Id {f3dd121e-604a-495b-ae98-29c9fcd2c0d9}
   Method Enable: Id {7ca4f60a-d1e0-4397-a83a-ed8dcb1017aa}
   Method Finish: Id {5b10ef5d-aac9-4514-b56a-99e09c68d7d2}
   Method Init: Id {10e2e475-1124-4c32-9d48-21872f6d1b74}
   Property InstanceCtrl: Id {7acdd1cc-198f-40bb-ba40-7856faf0d91c}
   Set Set: Id {2d3d313b-7311-479e-b918-28346a8bce77}
   Property InstanceState: Id {c2466ee2-4a57-4083-9c87-9e9f7eba2a74}
   Set Set: Id {e5a17682-314e-4e49-9b97-297ce85960e3}
   Method ListData: Id {8b730337-4e4b-4900-b4e8-13a7fa236b19}
   Property MessageLevel: Id {8ade6450-90c5-4683-b47c-6063ab1cfae3}
   Get Get: Id {b8718ada-c11b-4f81-b30a-3da434a9b4eb}
   Set Set: Id {16f6be41-bbda-46b4-a576-479cb4060503}
   Method Proceed: Id {f9a2f6e2-08f8-408b-a37e-4b3a16a77892}
   Property ProcessLinkedLists: Id {841e2785-8a81-4dab-ab69-a2404506471d}
   Set Set: Id {df60a9ec-7446-4a8a-92e2-3d5f72426dde}
   Property State: Id {257b9e36-771d-4714-8e16-430670e6fe24}
   Set Set: Id {588232c9-69de-48cc-813f-9f958d7bf6a6}
   Method Work: Id {c9245136-972a-4403-803b-e5d1ec9271e9}
   Property WriteTimeVariant: Id {741bcc54-9ee2-4811-8354-d070bf4ab52f}
   Get Get: Id {10a241a2-b4c9-46fa-b817-d2141a3ed1bb}
   Set Set: Id {a4dacca1-c32a-41f0-a14c-c44274b906db}
   Property XtsTransportCtrl: Id {3391bec1-98d1-4039-b0cc-fd4068165ffc}
   Set Set: Id {4fe1f55c-1a91-41e0-ad15-d1076bfbadce}
   Property XtsTransportState: Id {fa356716-e420-4889-891d-40c9f915f287}
   Set Set: Id {caa6f3cc-431a-488e-b079-3523f2bff879} *)
